FUNCTION_BLOCK FB_IndexedSiliconeMachine
VAR

    // =====================================================
    // CORE COMPONENTS
    // =====================================================
    fbIndex                     : FB_IndexTable4;
    fbMainDoorLock              : FB_MainDoorLock;
    fbNestManager               : FB_NestTableManager;
    fbOperatorStation           : FB_OperatorStation;
    

    // =====================================================
    // PROCESS COMPONENTS
    // =====================================================
    fbProcessStation            : FB_ProcessStation;
    fbProcessCycle              : FB_ProcessCycle;

    fbSiliconeProcess           : FB_SiliconeProcess;
    fbAssemblyStation           : FB_AssemblyStation;

    fbIvek                      : FB_IvekDigiSpense4000;
    fbIvekSettingsLauncher      : FB_IvekSettingsLauncher;

    ipEquipment                 : I_ProcessEquipment;

	// =====================================================
    // SILICONE SUPPLY 
    // =====================================================
	fbSiliconeSupply       : FB_SiliconeSupplySystem;
	stSiliconeSupplyStatus : ST_SiliconeSupplyStatus;
	stSiliconeSupplyConfig : ST_SiliconeSupplyConfig;
	
    // =====================================================
    // SUPPORT COMPONENTS
    // =====================================================
    fbSiliconeSupportCylinder   : FB_Support;
    fbAssemblySupportCylinder   : FB_Support;

    // =====================================================
    // MACHINE MODES
    // =====================================================
    fbManualMode                : FB_ManualMode;
	bManualAssemblySupportRaised : BOOL;

    // =====================================================
    // MACHINE / CYCLE STATES
    // =====================================================
    eMachineState               : E_MachineState := E_MachineState.PowerUp;
    ePreviousMachineState       : E_MachineState := E_MachineState.PowerUp;
    eCycleState                 : E_CycleState := E_CycleState.Disabled;

    bMachineStateEntry          : BOOL;

    eInitialisingWaitReason     : E_InitialisingWaitReason :=
                                    E_InitialisingWaitReason.None;

    eStoppingWaitReason         : E_StoppingWaitReason :=
                                    E_StoppingWaitReason.None;

    // =====================================================
    // NEST DATA
    // =====================================================
    stOperatorNest              : ST_Nest;
    stSiliconeNest              : ST_Nest;
    stAssemblyNest              : ST_Nest;
    stProcessNest               : ST_Nest;
	stFaultNest 				: ST_Nest;

    stLastResult                : ST_ProcessResult;
	bDisabledNestPartPresent 	: BOOL;

    // =====================================================
    // COMPONENT STATUS
    // =====================================================
    stOperatorStatus            : ST_OperatorStationStatus;
    stIndexStatus               : ST_IndexStatus;
    stProcessStationStatus      : ST_ProcessStationStatus;
    stAssemblyStationStatus     : ST_AssemblyStationStatus;
    stMainDoorLockStatus        : ST_MainDoorLockStatus;
	uiResetStatisticsNestIdOld 	: UINT;
	

    // =====================================================
    // MACHINE PERMISSIVES / OUTPUTS
    // =====================================================
    stPermissives               : ST_MachinePermissives;
    stOutputsInternal           : ST_MachineOutputs;
	stFaultRejectResult 		: ST_ProcessResult;
    // =====================================================
    // PROCESS CYCLE INTERFACE
    // =====================================================
    stProcessCycleInputs        : ST_ProcessCycleInputs;
    stProcessCycleRequests      : ST_ProcessCycleRequests;
    stProcessCycleStatus        : ST_ProcessCycleStatus;

    // =====================================================
    // MANUAL MODE INTERFACE
    // =====================================================
    stManualModeInputs          : ST_ManualModeInputs;
    stManualModeRequests        : ST_ManualModeRequests;
    stManualModeStatus          : ST_ManualModeStatus;

    // =====================================================
    // SUPPORT COMMANDS
    // =====================================================
    bSiliconeSupportRaiseRequest  : BOOL;
    bSiliconeSupportLowerRequest  : BOOL;

    bAssemblySupportRaiseRequest  : BOOL;
    bAssemblySupportLowerRequest  : BOOL;

    // =====================================================
    // INDEX COMMAND / FEEDBACK
    // =====================================================
    bManualIndexRequestAccepted             : BOOL;
    bManualAssemblyCycleActive                : BOOL;
    bManualSiliconeCycleActive                 : BOOL;
    bIndexRequestAcceptedFeedback           : BOOL;
    bIndexRecoveryRequestAcceptedFeedback   : BOOL;

    bIndexStable                            : BOOL;
    bIndexDone                              : BOOL;

    // =====================================================
    // PROCESS COMMAND / FEEDBACK
    // =====================================================
    bProcessStartPulse            : BOOL;
    bProcessReady                 : BOOL;
    bResultStoredFeedback         : BOOL;
    bIvekOperationPermissive      : BOOL;
    bIvekMaintenancePermissive    : BOOL;
    bIvekOperationalHealthy       : BOOL;
    bIvekAutoCycleReady           : BOOL;
    bIvekUnexpectedNotReady       : BOOL;
    tonIvekInitialisingRecovery   : TON;
    tonIvekReferenceStable        : TON;
    tonIvekUnexpectedNotReady     : TON;
    tonIvekCommunicationStop      : TON;
    tonIvekReferenceStop          : TON;

    bProcExtend                   : BOOL;
    bProcRetract                  : BOOL;

	bSiliconeProcessPartVacuumEnable : BOOL;
	bPartVacuumReleasePending        : BOOL;
	bSiliconeProcessAirEnable 		 : BOOL;
    // =====================================================
    // INITIALISATION / STOPPING
    // =====================================================
    bInitialisationComplete       : BOOL;
    bStoppingComplete             : BOOL;

    bInitialisationTimeoutFault   : BOOL;
    bStoppingTimeoutFault         : BOOL;
	bStopRequestTimeout 		  : BOOL;
	
	bExtractorAutoCycleFault 	  : BOOL;
	
    tonInitialising               : TON;
	tonInitialisingMinTime 	      : TON;
    tonStopping                   : TON;
    tonAutoCycleIdleTimeout       : TON;
	tonMainDoorNotClosed 		  : TON;
	tonStopRequest 				  : TON;
	
	
	bStopRequested 				  : BOOL;
    // =====================================================
    // AIR / DOOR CONTROL
    // =====================================================
    bAirAndDoorEnable             : BOOL;
    bAirSupplyLatched             : BOOL;
    bAirSupplyEnable              : BOOL;

    // =====================================================
    // SAFETY / FAULT HANDLING
    // =====================================================
    bSafetyDropRequest            : BOOL;

    fbEventFaultTrigger           : R_TRIG;
    fbResetTrigger                : R_TRIG;
	bFaultResetRequested 		  : BOOL;

    tpSafetyRunDrop               : TP;
	bHmiLogoutFault 				: BOOL;
		
	bSiliconePressureFault 			: BOOL;
	bNozzlePressureFault   			: BOOL;

	bSiliconePressureConfigRequired : BOOL;
	bNozzlePressureConfigRequired   : BOOL;
    // =====================================================
    // CONFIGURATION
    // =====================================================
    bConfigured                   : BOOL;
	
	// =====================================================
    // LEDS
    // =====================================================
	eMode_LED_Start 				: E_LEDs_Mode := E_LEDs_Mode.OFF;
	eMode_LED_Reset 				: E_LEDs_Mode := E_LEDs_Mode.OFF;
	eMode_LED_PASS  				: E_LEDs_Mode := E_LEDs_Mode.OFF;
	eMode_LED_Fail  				: E_LEDs_Mode := E_LEDs_Mode.OFF;

	tonLedBlink    					: TON;
	bLedBlink      					: BOOL;
	fbLedBlinkTrigger 				: R_TRIG;
	bLedBlinkState 					: BOOL;
	
	uiHistoryNestId 				: UINT;
	bHistoryPassed  				: BOOL;
	stHistoryNest   				: ST_Nest;
	// =====================================================
    // Extractor
    // =====================================================
	bExtractorEnable 				: BOOL;
	
	// CSV cycle data
	stCycleDataCSV      			: ST_CycleDataCSV;
	bCycleDataCSVWrite  			: BOOL;

END_VAR

METHOD CheckComponentFaults : BOOL
// =========================================================
// COMPONENT FAULT AGGREGATION
// =========================================================

CheckComponentFaults := FALSE;

IF fbMainDoorLock.IsFaulted()
    OR fbIndex.IsFaulted()
	OR fbSiliconeSupportCylinder.IsFaulted()
	OR fbAssemblySupportCylinder.IsFaulted()
    OR fbAssemblyStation.IsFaulted()
    OR fbProcessStation.IsFaulted()

    // Enable after equipment commissioning.
    // OR ipEquipment.IsFaulted()
THEN

    bSafetyDropRequest := TRUE;
    eMachineState := E_MachineState.Fault;

    CheckComponentFaults := TRUE;

END_IF
END_METHOD

METHOD PUBLIC Cyclic
VAR_INPUT
    stInputs       : ST_MachineInputs;
    stCommand      : ST_MachineCommand;
    stConfig       : ST_MachineConfig;
    stIvekInput    : ST_IvekCyclicInput;
    bIvekCommsOk   : BOOL;
	blogoutHMI	   : BOOL;

	
END_VAR
VAR_OUTPUT
    stOutputs      : ST_MachineOutputs;
    stStatus       : ST_MachineStatus;
    stIvekOutput   : ST_IvekCyclicOutput;
	stCycleDataCSVOut     : ST_CycleDataCSV;
	bCycleDataCSVWriteOut : BOOL;
END_VAR
// =========================================================
// GLOBAL MACHINE FAULT CONDITION
// =========================================================
// Any loss of the validated TwinSAFE safety status must place
// the machine in Fault immediately, regardless of machine state.
// =========================================================

IF NOT stInputs.stSafety.bSafetyOk OR bSafetyDropRequest THEN

    eMachineState := E_MachineState.Fault;

END_IF

// =========================================================
// MACHINE STOP REQUEST LATCH
// =========================================================

// Memorise the Stop command until the machine has
// completed the required stopping sequence.
IF (stCommand.bStop OR stCommand.bPowerDownRequest)
    AND (eMachineState <> E_MachineState.Stopping)
    AND (eMachineState <> E_MachineState.Stopped)
THEN
    bStopRequested := TRUE;
END_IF

// =========================================================
// LED BLINK GENERATOR
// =========================================================

tonLedBlink(
    IN := NOT tonLedBlink.Q,
    PT := T#500MS
);

fbLedBlinkTrigger(
    CLK := tonLedBlink.Q
);

IF fbLedBlinkTrigger.Q THEN
    bLedBlinkState := NOT bLedBlinkState;
END_IF

bLedBlink := bLedBlinkState;
// =========================================================
// DETERMINISTIC CYCLIC INITIALISATION
// =========================================================

// Deterministic defaults
ResetCyclicOutputs();

// CSV write request is generated for one PLC scan
bCycleDataCSVWrite := FALSE;

// This request is generated for one PLC scan by an internal machine fault.
// The TP converts the one-scan request into the required TwinSAFE run-drop time.
bSafetyDropRequest := FALSE;
bMachineStateEntry := eMachineState <> ePreviousMachineState;
ePreviousMachineState := eMachineState;
fbResetTrigger(
    CLK := stCommand.bReset
);

IF fbResetTrigger.Q THEN
    fbSiliconeProcess.RequestReset();
    fbAssemblyStation.RequestReset();
END_IF

fbSiliconeSupply.Cyclic(
    bLevel1Ok := stInputs.bSiliconeMinimumLevel1,
    bLevel2Ok := stInputs.bSiliconeMinimumLevel2,
    rSiliconePressureBar := stInputs.rSiliconePressureBar,
    rNozzlePressureBar := stInputs.rNozzlePressureBar,
    rVacuumEngineering := stInputs.rVacuumEngineering,

    stConfig := GVL_Config.stMachine.stSiliconeSupply,

    bCmdSelectReservoir1 := GVL_SiliconeSupply_Interface.bCmdSelectReservoir1,
    bCmdSelectReservoir2 := GVL_SiliconeSupply_Interface.bCmdSelectReservoir2,
    bCmdStartDegassing1 := GVL_SiliconeSupply_Interface.bCmdStartDegassing1,
    bCmdStartDegassing2 := GVL_SiliconeSupply_Interface.bCmdStartDegassing2,
    bCmdCancelDegassing := GVL_SiliconeSupply_Interface.bCmdCancelDegassing,
    bManualSelectionAllowed := eMachineState = E_MachineState.Stopped,

    bDispenseActive := fbSiliconeProcess.IsBusy() OR fbIvek.IsFluidicActive(),
    bDispenseValveRequest := fbSiliconeProcess.GetPinchValveRequest() OR fbIvek.IsFluidicActive(),
    bImmediateFault := eMachineState = E_MachineState.Fault,

    stPersistent := GVL_Persistent.stSiliconeSupply,

    bVacuumPump => stOutputsInternal.bVacuumPumpEnable,
    bVacuumToAir1 => stOutputsInternal.bVacuumAirSolenoid1,
    bVacuumToAir2 => stOutputsInternal.bVacuumAirSolenoid2,
    bPinchValve1 => stOutputsInternal.bSiliconePinchValve1,
    bPinchValve2 => stOutputsInternal.bSiliconePinchValve2
);

stSiliconeSupplyStatus := fbSiliconeSupply.GetStatus();
GVL_SiliconeSupply_Interface.stStatus := stSiliconeSupplyStatus;
stStatus.stSiliconeSupply := stSiliconeSupplyStatus;

IF fbSiliconeSupply.HasStopRequest() THEN
    bStopRequested := TRUE;
END_IF

IF eMachineState = E_MachineState.AutoCycle
AND stSiliconeSupplyStatus.bReservoirSelectionRequired THEN
    bStopRequested := TRUE;
END_IF

// Loss of IVEK reference is a recoverable stop condition, not an Immediate
// Fault. Stop the active machine and require Engineer Reference in Settings.
IF fbIvek.IsReferenceRequired()
AND (eMachineState = E_MachineState.AutoCycle OR eMachineState = E_MachineState.Manual) THEN
    bStopRequested := TRUE;
END_IF

// The Assembly Station is executed with its physical I/O in the component section below.

bProcessStartPulse := FALSE;

// Automatic door-lock request. Air supply is managed independently by the machine states below.
bAirAndDoorEnable := (eMachineState = E_MachineState.Initialising) OR (eMachineState = E_MachineState.ReadyToStart) OR (eMachineState = E_MachineState.AutoCycle) OR (eMachineState = E_MachineState.Manual);

stIndexStatus := fbIndex.GetStatus();
bIndexStable := NOT stIndexStatus.bBusy AND stInputs.bIndexReady AND stInputs.bIndexLocked AND stInputs.eIndexPosition <> E_TablePosition.Unknown;
bIndexDone := fbIndex.IsDone();

// =========================================================
// HMI LOGOUT SUPERVISION
// =========================================================
//
// If the HMI heartbeat is lost while the machine is already
// Stopped, the machine must remain Stopped.
//
// If the heartbeat is lost in any other operating state,
// the machine enters Fault immediately.
//
// Fault is never overridden by the HMI logout condition.
// =========================================================


// Loss of HMI heartbeat also requests a controlled stop.
// Fault has higher priority and is handled separately.
IF blogoutHMI
    AND (eMachineState = E_MachineState.Stopped OR eMachineState = E_MachineState.Stopping)THEN
	bStopRequested := TRUE;
	
ELSIF blogoutHMI
    AND (eMachineState <> E_MachineState.Stopped AND eMachineState <> E_MachineState.Stopping)THEN 
	bHmiLogoutFault := TRUE;
    bSafetyDropRequest := TRUE;
END_IF




// =========================================================
// PROCESS EQUIPMENT CONFIGURATION / CYCLIC EXECUTION
// =========================================================

// Configure the real IVEK process equipment once.
IF NOT bConfigured THEN

    ipEquipment := fbIvek;

    fbProcessStation.Configure(
        ipNewEquipment := ipEquipment
    );

    bConfigured := TRUE;

END_IF


// ---------------------------------------------------------
// IVEK machine-level operation permissive
// ---------------------------------------------------------
// Runtime motion is allowed only while:
// - EtherNet/IP communication is healthy;
// - process safety is permitted;
// - machine air is validated;
// - the machine is in AutoCycle or Manual;
// - the machine is not in Fault.
//
// FB_IvekDigiSpense4000 performs the controlled Stop-before-
// MotionDisable behaviour if this permissive is removed while
// Production is active.
bIvekOperationPermissive :=
    bIvekCommsOk
    AND stInputs.stSafety.bProcessSafetyPermitted
    AND GVL_Safety.bAirSupplySafe
    AND eMachineState <> E_MachineState.Fault
    AND (
        eMachineState = E_MachineState.Initialising
        OR eMachineState = E_MachineState.ReadyToStart
        OR eMachineState = E_MachineState.AutoCycle
        OR eMachineState = E_MachineState.Manual
    );

// Engineer Settings operations are only permitted while Stopped with the
// process safety circuit and pneumatic supply healthy.
bIvekMaintenancePermissive :=
    bIvekCommsOk
    AND (eMachineState = E_MachineState.Stopped)
    AND stInputs.stSafety.bProcessSafetyPermitted
    AND GVL_Safety.bAirSupplySafe
    AND stInputs.bMainDoorClosed;
	
stStatus.bIvekClearFaultPermissive :=
    bIvekCommsOk
    AND (eMachineState = E_MachineState.Stopped OR eMachineState = E_MachineState.Fault)
    AND fbIvek.IsFaulted();


// Always execute the real IVEK object for communication diagnostics,
// even while process simulation is selected.
fbIvek.stCyclicIn := stIvekInput;
fbIvek.bCommunicationOk := bIvekCommsOk;
fbIvek.bOperationPermissive := bIvekOperationPermissive;
fbIvek.bSystemInitialising := (eMachineState = E_MachineState.Initialising);
fbIvek.bMaintenancePermissive := bIvekMaintenancePermissive;
fbIvek.bPrimePermissive :=
    (eMachineState = E_MachineState.Manual)
    AND bIvekCommsOk
    AND stInputs.stSafety.bProcessSafetyPermitted
    AND GVL_Safety.bAirSupplySafe;
fbIvek.Cyclic();

// =========================================================
// IVEK OPERATIONAL INTERLOCK
// =========================================================
// ReadyProduction is expected to drop during a valid dispense, therefore
// permanent health is evaluated separately from start readiness.
bIvekOperationalHealthy :=
    bIvekCommsOk
    AND NOT fbIvek.IsFaulted()
    AND NOT fbIvek.IsReferenceRequired();

bIvekAutoCycleReady :=
    bIvekOperationalHealthy
    AND fbIvek.bReadyProduction
    AND NOT fbIvek.IsFluidicActive()
    AND NOT fbIvek.IsReferenceActive();

// ReadyProduction=FALSE is abnormal only while the process is idle.
// This avoids treating a normal dispense as "not ready".
bIvekUnexpectedNotReady :=
    bIvekOperationalHealthy
    AND (eMachineState <> E_MachineState.Initialising)
    AND NOT fbIvek.bReadyProduction
    AND NOT fbIvek.IsBusy()
    AND NOT fbSiliconeProcess.IsBusy()
    AND NOT fbIvek.IsFluidicActive()
    AND NOT fbIvek.IsReferenceActive();

// ReadyProduction can briefly drop around a legitimate Production transition.
// Do not stop the whole machine on a one-scan / short transient.
// Communication loss, IVEK Fault and Reference Required remain immediate
// operational-stop conditions through bIvekOperationalHealthy.
// Transient IVEK conditions must not stop the machine immediately.
// Actual IVEK faults remain immediate; communication, reference-required
// and generic not-ready are debounced to tolerate short status gaps.
tonIvekUnexpectedNotReady(
    IN := bIvekUnexpectedNotReady,
    PT := T#3S
);

tonIvekCommunicationStop(
    IN := NOT bIvekCommsOk
        AND (
            eMachineState = E_MachineState.ReadyToStart
            OR eMachineState = E_MachineState.AutoCycle
            OR eMachineState = E_MachineState.Manual
        ),
    PT := T#2S
);

tonIvekReferenceStop(
    IN := bIvekCommsOk
        AND fbIvek.IsReferenceRequired()
        AND (
            eMachineState = E_MachineState.ReadyToStart
            OR eMachineState = E_MachineState.AutoCycle
            OR eMachineState = E_MachineState.Manual
        ),
    PT := T#2S
);

// Engineer Settings commands. HMI page access is Engineer-only; PLC also
// enforces Stopped + safety/air conditions before the FB accepts motion.
// Controlled IVEK stop before PLC shutdown or reboot.
IF stCommand.bIvekMaintenanceStop THEN
    fbIvek.RequestStop();
END_IF

IF stCommand.bPowerDownRequest THEN

    // Stop active equipment/process sequences before PLC shutdown or reboot.
    fbIvek.RequestStop();
    fbSiliconeProcess.RequestStop();
    fbAssemblyStation.RequestStop();
	bStopRequested := TRUE;

END_IF

IF stCommand.bIvekReference THEN
    fbIvek.RequestReference();
END_IF

IF stCommand.bIvekClearFault THEN
    fbIvek.RequestReset();
END_IF



// Process simulation removed from runtime path. The real IVEK is always used.


IF stCommand.usiRecipeRequest <> 0 THEN
    ipEquipment.SetRecipe(stCommand.usiRecipeRequest);
END_IF


// =========================================================
// SILICONE PROCESS COORDINATOR
// =========================================================
// Execute exactly once per PLC scan, after the selected process
// equipment has updated its status for this scan.
fbSiliconeProcess.Cyclic(
    bSupplyReady 				:= fbSiliconeSupply.IsReadyForDispense(),
    bEquipmentReady 			:= fbIvek.IsReady(),
    bEquipmentBusy 				:= fbIvek.IsBusy(),
    bEquipmentDone 				:= fbIvek.IsDone(),
    bEquipmentFaulted 			:= fbIvek.IsFaulted(),
    stEquipmentResult 			:= fbIvek.GetResult(),
    bSiliconeSupportExtended 	:= stInputs.bSiliconeSupportExtended,
    bExtractorReady 			:= stPermissives.bExtractorReady,
	bPartVacuumOk 				:= stInputs.bPartVacuumOk,
	tPartVacuumBuildTimeout 	:= GVL_Config.stMachine.tPartVacuumBuildTimeout,
	tPartVacuumReleaseTimeout 	:= GVL_Config.stMachine.tPartVacuumReleaseTimeout,
    tPinchSettlingDelay 		:= GVL_Config.stMachine.stSiliconeSupply.tPinchValveSettlingDelay,
    tEquipmentStartTimeout 		:= GVL_Config.stMachine.stSiliconeSupply.tIvekStartTimeout,
    tEquipmentCompleteTimeout 	:= GVL_Config.stMachine.stSiliconeSupply.tIvekCompleteTimeout,
	bSiliconeStationPartPresent := stInputs.bSiliconeStationPartPresent,
    bPartVacuumEnable 			=> bSiliconeProcessPartVacuumEnable,
	bSiliconeAirEnable 			=> bSiliconeProcessAirEnable
);

// The coordinator generates one-scan equipment requests.
// The equipment object latches these requests and executes them
// on its next Cyclic() call.
IF fbSiliconeProcess.GetEquipmentStopRequest() THEN
    fbIvek.RequestStop();
END_IF

IF fbSiliconeProcess.GetEquipmentResetRequest() THEN
    fbIvek.RequestReset();
END_IF

IF fbSiliconeProcess.GetEquipmentStartRequest() THEN
    fbIvek.RequestStart();
END_IF

stStatus.rIvekHeaterTemperature :=
    stInputs.rIvekHeaterTemperature;

stStatus.bIvekHeaterTemperatureOutOfRange :=
    (stInputs.rIvekHeaterTemperature <
        GVL_Config.stMachine.stSiliconeSupply.rIvekHeaterTemperatureMin)
    OR
    (stInputs.rIvekHeaterTemperature >
        GVL_Config.stMachine.stSiliconeSupply.rIvekHeaterTemperatureMax);

stStatus.eIvekStatusState := fbIvek.GetStatusState();

// =========================================================
// NEST MANAGEMENT

fbNestManager.Cyclic(
    bIndexStable := bIndexStable,
    bIndexComplete := bIndexDone,

    eIndexPosition := stInputs.eIndexPosition,

    bGearboxAssemblyPartPresent := stInputs.bGearboxAssemblyPartPresent,
    bReservoirPartPresent := stInputs.bReservoirPartPresent,
    eOperatorPosition := stConfig.eOperatorPosition,
    bIndexSamePositionDetected := stIndexStatus.bSamePositionDetected,
    aNestEnabled := stConfig.aNestEnabled
);


stOperatorNest := fbNestManager.GetNestAtPosition(stConfig.eOperatorPosition);
stSiliconeNest := fbNestManager.GetNestAtPosition(stConfig.eSiliconePosition);
stAssemblyNest := fbNestManager.GetNestAtPosition(stConfig.eAssemblyPosition);

// =========================================================
// DISABLED OPERATOR NEST PART DETECTION
// =========================================================
// Disabled nests keep the existing machine behaviour while empty.
// If a part is physically detected at the operator station while
// the current operator nest is disabled, indexing will be inhibited.

bDisabledNestPartPresent :=
    NOT stOperatorNest.bEnabled
    AND
    (
        stInputs.bGearboxAssemblyPartPresent
        OR stInputs.bReservoirPartPresent
    );

// =========================================================
// MANUAL MODE - NEW PART / NEST RESULT RESET
// =========================================================
// A newly loaded part in Manual mode starts a new process history for
// the physical nest. Clear Silicone / Assembly / final results left by
// the previous part.
//
// AutoCycle keeps its existing PASS/FAIL disposition-based clear logic.
IF (eMachineState = E_MachineState.Manual)
AND stOperatorNest.bPartLoadedPulse THEN

    fbNestManager.ClearOperatorNest(
        ePosition := stConfig.eOperatorPosition
    );

    // Refresh the local snapshot after clearing the internal nest data.
    stOperatorNest :=
        fbNestManager.GetNestAtPosition(stConfig.eOperatorPosition);

END_IF

// =========================================================
// RESET CURRENT NEST STATISTICS
// =========================================================

IF stCommand.uiResetStatisticsNestId >= 1
    AND stCommand.uiResetStatisticsNestId <= 4
    AND stCommand.uiResetStatisticsNestId <> uiResetStatisticsNestIdOld
THEN

    fbNestManager.ResetNestStatistics(
        uiNestId := stCommand.uiResetStatisticsNestId
    );

END_IF

uiResetStatisticsNestIdOld :=stCommand.uiResetStatisticsNestId;

fbNestManager.CountStatisticsAtPosition(
    ePosition := stConfig.eOperatorPosition
);



// =========================================================
// TEST HISTORY EVENT
// =========================================================

IF fbNestManager.GetStatisticsEvent(
    uiNestId => uiHistoryNestId,
    bPassed  => bHistoryPassed
) THEN

    // Get the complete nest data at the moment
    // the result is added to the statistics.
    stHistoryNest := fbNestManager.GetNestAtPosition( stConfig.eOperatorPosition );


    // -----------------------------------------------------
    // STORE TEST HISTORY ENTRY
    // -----------------------------------------------------

    GVL_Persistent.astTestHistory[GVL_Persistent.uiTestHistoryWriteIndex].uiNestId 				:= uiHistoryNestId;
    GVL_Persistent.astTestHistory[GVL_Persistent.uiTestHistoryWriteIndex].eResult 				:= stHistoryNest.eDisposition;
    GVL_Persistent.astTestHistory[GVL_Persistent.uiTestHistoryWriteIndex].bSiliconeValid 		:= stHistoryNest.stSiliconeResult.bValid;
    GVL_Persistent.astTestHistory[GVL_Persistent.uiTestHistoryWriteIndex].bSiliconePass 		:= stHistoryNest.stSiliconeResult.bPassed;
    GVL_Persistent.astTestHistory[GVL_Persistent.uiTestHistoryWriteIndex].bAssemblyValid 		:= stHistoryNest.stAssemblyResult.bValid;
    GVL_Persistent.astTestHistory[GVL_Persistent.uiTestHistoryWriteIndex].bAssemblyPass 		:= stHistoryNest.stAssemblyResult.bPassed;
	GVL_Persistent.astTestHistory[GVL_Persistent.uiTestHistoryWriteIndex].sDate 				:= GVL_MASTER.sSystemDate;
	GVL_Persistent.astTestHistory[GVL_Persistent.uiTestHistoryWriteIndex].sTime 				:= GVL_MASTER.sSystemTime;
				
				// Final result text
		IF stHistoryNest.stResult.bPassed THEN
			GVL_Persistent.astTestHistory[GVL_Persistent.uiTestHistoryWriteIndex].sResult := 'PASS';
		ELSE
			GVL_Persistent.astTestHistory[GVL_Persistent.uiTestHistoryWriteIndex].sResult := 'FAIL';
		END_IF;
		
		
		// Silicone result text
		IF NOT stHistoryNest.stSiliconeResult.bValid THEN
		
			GVL_Persistent.astTestHistory[GVL_Persistent.uiTestHistoryWriteIndex].sSiliconeResult := 'NOT STARTED';
		
		ELSIF stHistoryNest.stSiliconeResult.bPassed THEN
		
			GVL_Persistent.astTestHistory[GVL_Persistent.uiTestHistoryWriteIndex].sSiliconeResult := 'PASS';
		
		ELSE
		
			GVL_Persistent.astTestHistory[GVL_Persistent.uiTestHistoryWriteIndex].sSiliconeResult := 'FAIL';
		
		END_IF;
		
		
		// Flipping result text
		IF NOT stHistoryNest.stAssemblyResult.bValid THEN
		
			GVL_Persistent.astTestHistory[GVL_Persistent.uiTestHistoryWriteIndex].sFlippingResult := 'NOT STARTED';
		
		ELSIF stHistoryNest.stAssemblyResult.bPassed THEN
		
			GVL_Persistent.astTestHistory[GVL_Persistent.uiTestHistoryWriteIndex].sFlippingResult := 'PASS';
		
		ELSE
		
			GVL_Persistent.astTestHistory[GVL_Persistent.uiTestHistoryWriteIndex].sFlippingResult := 'FAIL';
		
		END_IF;
				
		// -----------------------------------------------------
		// PREPARE CSV CYCLE DATA
		// -----------------------------------------------------
		
		stCycleDataCSV.uiNestId :=
			GVL_Persistent.astTestHistory[GVL_Persistent.uiTestHistoryWriteIndex].uiNestId;
		
		stCycleDataCSV.sGeneralResult :=
			GVL_Persistent.astTestHistory[GVL_Persistent.uiTestHistoryWriteIndex].sResult;
		
		stCycleDataCSV.sSiliconeResult :=
			GVL_Persistent.astTestHistory[GVL_Persistent.uiTestHistoryWriteIndex].sSiliconeResult;
		
		stCycleDataCSV.sFlippingResult :=
			GVL_Persistent.astTestHistory[GVL_Persistent.uiTestHistoryWriteIndex].sFlippingResult;
		
		stCycleDataCSV.sDate :=
			GVL_Persistent.astTestHistory[GVL_Persistent.uiTestHistoryWriteIndex].sDate;
		
		stCycleDataCSV.sTime :=
			GVL_Persistent.astTestHistory[GVL_Persistent.uiTestHistoryWriteIndex].sTime;
		
		bCycleDataCSVWrite := TRUE;	
				
				
				
		// -----------------------------------------------------
		// ADVANCE TEST HISTORY WRITE INDEX
		// -----------------------------------------------------
		
		IF GVL_Persistent.uiTestHistoryCount < 2001 THEN
			GVL_Persistent.uiTestHistoryCount := GVL_Persistent.uiTestHistoryCount + 1;
		END_IF
		
		IF GVL_Persistent.uiTestHistoryWriteIndex < 2000 THEN
		
			GVL_Persistent.uiTestHistoryWriteIndex := GVL_Persistent.uiTestHistoryWriteIndex + 1;
		
		ELSE
		
			GVL_Persistent.uiTestHistoryWriteIndex := 0;
		
		END_IF
		

END_IF



// =========================================================
// OPERATOR STATION CONTROL
// =========================================================


// Operator exchange is evaluated independently of process-equipment implementation.
fbOperatorStation.Cyclic(
    bAutomaticActive := eMachineState = E_MachineState.AutoCycle,
    bIndexStable := bIndexStable,
    stOperatorNest := stOperatorNest,
    bGearboxAssemblyPartPresent := stInputs.bGearboxAssemblyPartPresent,
    bReservoirPartPresent := stInputs.bReservoirPartPresent,
    bRejectChutePartPresent := stInputs.bRejectChutePartPresent,
    bRequireRejectConfirm := stConfig.bRequireRejectConfirm,
    bAllowEmptyNestIndex := stConfig.bAllowEmptyNestIndex);
	
stOperatorStatus := fbOperatorStation.GetStatus();

// =========================================================
// OPERATOR NEST RESULT RELEASE
// =========================================================


// PASS: clear after part removal.
IF stOperatorNest.stResult.bValid
    AND stOperatorNest.stResult.bPassed
    AND stOperatorStatus.bPartRemovedConfirmed
THEN

    fbNestManager.ClearOperatorNest(
        stConfig.eOperatorPosition
    );

END_IF


// FAIL: clear only after reject confirmation.
IF stOperatorNest.stResult.bValid
    AND NOT stOperatorNest.stResult.bPassed
    AND stOperatorStatus.bRejectConfirmed
THEN

    fbNestManager.ClearOperatorNest(
        stConfig.eOperatorPosition
    );

END_IF

// =========================================================
// MACHINE PERMISSIVE AGGREGATION
// =========================================================

// Explicit permissive aggregation.
stPermissives.bSafetyIndexPermissive 	:= 	stInputs.stSafety.bMotionSafetyPermitted;
stPermissives.bOperatorIndexPermissive 	:= 	fbOperatorStation.IndexPermissive();
stPermissives.bProcessIndexPermissive 	:= 	NOT fbSiliconeProcess.IsBusy()
											AND NOT fbSiliconeProcess.IsFaulted()
											AND fbAssemblyStation.IndexPermissive();

stPermissives.bIndexMoveAllowed :=
											stPermissives.bSafetyIndexPermissive
											//AND stPermissives.bOperatorIndexPermissive
											AND stPermissives.bProcessIndexPermissive
											AND NOT bDisabledNestPartPresent;


stPermissives.bProcessStartAllowed 		:= 	stInputs.stSafety.bProcessSafetyPermitted
											AND stInputs.bIndexReady
											AND stInputs.bIndexLocked
											AND stInputs.bReservoirPartPresent;
											
stPermissives.bExtractorReady 			:=  stInputs.bExtractorRunning;


// =========================================================
// INITIALISATION PERMISSIVES
// =========================================================

stPermissives.bAirSupplyReady :=
	GVL_Safety.bAirSupplySafe;

stPermissives.bSiliconeSupportHome :=
    stInputs.bSiliconeSupportRetracted;

stPermissives.bAssemblySupportHome :=
    stInputs.bAssemblySupportRetracted;

stPermissives.bSupportsHome :=
    stPermissives.bSiliconeSupportHome
    AND stPermissives.bAssemblySupportHome;

stPermissives.bAssemblyStationHome := fbAssemblyStation.IsHome();

stPermissives.bIndexInitialisationReady :=
    ( NOT stIndexStatus.bBusy
        OR
        (stIndexStatus.eState = E_IndexState.WrongPositionRecovery
            AND stInputs.eIndexPosition = E_TablePosition.Unknown)
    )
    AND NOT fbIndex.IsFaulted();

stPermissives.bDoorInitialisationReady :=
    NOT fbMainDoorLock.IsFaulted()
    AND fbMainDoorLock.IsReadyForAutomatic();

stPermissives.bInitialisationAllowed :=
    stInputs.stSafety.bSafetyOk
    AND stPermissives.bAirSupplyReady
    AND stPermissives.bIndexInitialisationReady
    AND stPermissives.bSupportsHome
    AND stPermissives.bAssemblyStationHome
    AND NOT fbAssemblyStation.IsFaulted()
    AND stPermissives.bDoorInitialisationReady
    AND stPermissives.bExtractorReady
    AND NOT stInputs.bIvekHeaterControllerAlarm
	AND NOT stStatus.bIvekHeaterTemperatureOutOfRange ;
	//AND stSiliconeSupplyStatus.bSiliconePressureOk
    //AND stSiliconeSupplyStatus.bNozzlePressureOk;
	

// =========================================================
// IVEK NATIVE SETTINGS LAUNCHER
// =========================================================
 
fbIvekSettingsLauncher(
    bOpenRequest 		:= GVL_HMI.bCmdOpenIvekSettings,
    bMachineStopped 	:= eMachineState = E_MachineState.Stopped,
    udiLauncherHeartbeat := GVL_HMI.udiIvekSettingsHeartbeat,
    bResetError 		:= stCommand.bReset,
    bLauncherActive 	:= GVL_HMI.bIvekSettingsActive,
    bOpenPermitted 		=> GVL_HMI.bIvekSettingsAccessAllowed,
    bSettingsInterlock 	=> GVL_HMI.bIvekSettingsInterlock,
    bLaunchPending 		=> GVL_HMI.bIvekSettingsLaunchPending,
    bLaunchBusy 		=> GVL_HMI.bIvekSettingsLaunchBusy,
    bLaunchError 		=> GVL_HMI.bIvekSettingsLaunchError,
    nLaunchErrorId 		=> GVL_HMI.nIvekSettingsLaunchErrorId,
    bActivationTimeout 	=> GVL_HMI.bIvekSettingsActTimeout,
    bHeartbeatLost 		=> GVL_HMI.bIvekSettingsHeartbeatLost
);

// =========================================================
// EVENT ARCHITECTURE NOTES
// =========================================================

// Event architecture from the Leak Tester.
// Point classification is fixed in PRG_Events; station latches are provided
// through stInputs.bEventFault and stInputs.bEventCycleStopRequest.

// =========================================================
// MANUAL MODE COORDINATOR
// =========================================================

// Manual-mode coordinator consumes only normalized component status and produces requests.
stManualModeInputs.bSafetyOk 						:= stInputs.stSafety.bSafetyOk;
stManualModeInputs.bMotionSafetyPermitted 			:= stInputs.stSafety.bMotionSafetyPermitted;
stManualModeInputs.bTwoHandsSafe 					:= stInputs.bTwoHandsSafe;
stManualModeInputs.bProcessSafetyPermitted 			:= stInputs.stSafety.bProcessSafetyPermitted;
stManualModeInputs.bMainDoorSafe 					:= stInputs.stSafety.bMainDoorSafe;
stManualModeInputs.bIndexReady 						:= stInputs.bIndexReady;
stManualModeInputs.bIndexLocked 					:= stInputs.bIndexLocked;
stManualModeInputs.bIndexBusy 						:= stIndexStatus.bBusy;
stManualModeInputs.bIndexFaulted 					:= fbIndex.IsFaulted();
stManualModeInputs.bSiliconeSupportExtended 		:=stInputs.bSiliconeSupportExtended;
stManualModeInputs.bSiliconeSupportRetracted 		:=stInputs.bSiliconeSupportRetracted;
stManualModeInputs.bAssemblySupportExtended 		:=stInputs.bAssemblySupportExtended;
stManualModeInputs.bAssemblySupportRetracted 		:=stInputs.bAssemblySupportRetracted;



stManualModeInputs.bProcessStationFaulted := fbProcessStation.IsFaulted();
stManualModeInputs.bEquipmentReady := fbIvek.IsReady();
stManualModeInputs.bEquipmentBusy := fbIvek.IsBusy();
stManualModeInputs.bEquipmentFaulted := fbIvek.IsFaulted();

stManualModeInputs.bIvekEnabled := bIvekCommsOk AND NOT fbIvek.bMotionDisabled;
stManualModeInputs.bIvekFluidicReady := fbIvek.IsFluidicReady();
stManualModeInputs.bIvekFluidicActive := fbIvek.IsFluidicActive();
stManualModeInputs.bPartVacuumOk := stInputs.bPartVacuumOk;
stManualModeInputs.bIvekPrimeEnable :=stCommand.bIvekPrimeEnable;
stManualModeInputs.bNozzlePressureOk :=stSiliconeSupplyStatus.bNozzlePressureOk;

stManualModeInputs.bSiliconeProcessReady := fbSiliconeProcess.IsReady();
stManualModeInputs.bSiliconeProcessBusy := fbSiliconeProcess.IsBusy();
stManualModeInputs.bSiliconeProcessFaulted := fbSiliconeProcess.IsFaulted();
stManualModeInputs.bSiliconeNestPartPresent := stSiliconeNest.bPartComplete;
stManualModeInputs.bSiliconeNestAlreadyProcessed :=
    stSiliconeNest.stSiliconeResult.bValid;

stManualModeInputs.bReservoirPartPresent :=stInputs.bSiliconeStationPartPresent;
stManualModeInputs.bAssemblyStationReady := fbAssemblyStation.IsReady();
stManualModeInputs.bAssemblyStationBusy := fbAssemblyStation.IsBusy();
stManualModeInputs.bAssemblyStationFaulted := fbAssemblyStation.IsFaulted();
stManualModeInputs.bAssemblyNestPartPresent := stAssemblyNest.bPartComplete;
stManualModeInputs.bAssemblyNestSiliconized :=
    stAssemblyNest.stSiliconeResult.bValid
    AND stAssemblyNest.stSiliconeResult.bPassed;
stManualModeInputs.bAssemblyNestAlreadyAssembled :=
    stAssemblyNest.stAssemblyResult.bValid;

fbManualMode.Cyclic(
    bEnable := eMachineState = E_MachineState.Manual,
    bStopRequest := bStopRequested,
    stCommand := stCommand,
    stInputs := stManualModeInputs,
    stRequests => stManualModeRequests,
    stStatus => stManualModeStatus);
	
	
// =========================================================
// SILICONE AIR OUTPUT ARBITRATION
// =========================================================

stOutputsInternal.bSiliconeAirEnable :=
    bSiliconeProcessAirEnable
    OR (
        (eMachineState = E_MachineState.Manual)
        AND stManualModeRequests.bSiliconeAirEnable
    );
	
	
// =========================================================
// PART VACUUM RELEASE CONFIRMATION
// =========================================================

// Latch the release condition when a process has finished
// while vacuum is still present, or when Manual Prime
// explicitly requests vacuum release.
IF (fbSiliconeProcess.IsDone() AND stInputs.bPartVacuumOk)
    OR stManualModeRequests.bPartVacuumReleaseRequest
THEN
    bPartVacuumReleasePending := TRUE;
END_IF

// Release is complete only after the Silicone Support is
// fully retracted and the station is confirmed empty.
IF bPartVacuumReleasePending
    AND stInputs.bSiliconeSupportRetracted
    AND NOT stInputs.bSiliconeStationPartPresent
THEN
    bPartVacuumReleasePending := FALSE;
END_IF

// A new intentional Manual Prime vacuum request is allowed
// only after the previous release sequence has physically
// completed.
IF (eMachineState = E_MachineState.Manual)
    AND stManualModeRequests.bPartVacuumEnable
    AND stInputs.bSiliconeSupportExtended
    AND stInputs.bSiliconeStationPartPresent
THEN
    bPartVacuumReleasePending := FALSE;
END_IF	
// Allow a new Silicone process to take ownership of the vacuum
// once a new part is confirmed in the raised Silicone Support.

IF bSiliconeProcessPartVacuumEnable
    AND stInputs.bSiliconeSupportExtended
    AND stInputs.bSiliconeStationPartPresent
THEN
    bPartVacuumReleasePending := FALSE;
END_IF
	
// =========================================================
// PART VACUUM OUTPUT ARBITRATION
// =========================================================
// In automatic operation the part vacuum follows the machine
// pneumatic lifecycle while the Silicone Support is retracted.
//
// During the Silicone process, FB_SiliconeProcess owns the vacuum.
// After dispensing it removes its vacuum request before the
// Silicone Support retracts. Once the support is fully retracted,
// the normal vacuum request is restored.
//
// Manual Mode keeps its existing independent vacuum control.

stOutputsInternal.bPartVacuumEnable :=
    NOT bPartVacuumReleasePending
    AND
    (
        bSiliconeProcessPartVacuumEnable
        OR (
            bExtractorEnable
            AND stInputs.bSiliconeSupportRetracted
        )
        OR (
            (eMachineState = E_MachineState.Manual)
            AND stManualModeRequests.bPartVacuumEnable
        )
    );
// Manual Prime equipment request.
// The complete mechanical/vacuum sequence is coordinated by FB_ManualMode.
IF (eMachineState = E_MachineState.Manual)
AND stManualModeRequests.bIvekPrime THEN
    fbIvek.RequestPrime();
END_IF

stProcessCycleInputs.bSiliconeSupportExtended := stInputs.bSiliconeSupportExtended;
stProcessCycleInputs.bSiliconeSupportRetracted := stInputs.bSiliconeSupportRetracted;
stProcessCycleInputs.bAssemblySupportExtended := stInputs.bAssemblySupportExtended;
stProcessCycleInputs.bAssemblySupportRetracted := stInputs.bAssemblySupportRetracted;

// =========================================================
// STOP REQUEST TIMEOUT SUPERVISION
// =========================================================
// Once a Stop request has been latched, the machine must
// reach the Stopping state within the allowed time.
//
// This supervises the conditions that may delay leaving
// AutoCycle or Manual mode after a Stop request.
tonStopRequest(
    IN := bStopRequested
        AND eMachineState <> E_MachineState.Stopping
        AND eMachineState <> E_MachineState.Stopped
        AND eMachineState <> E_MachineState.Fault,
    PT := T#10S
);

IF tonStopRequest.Q THEN
    bStopRequestTimeout := TRUE;
    bSafetyDropRequest := TRUE;
END_IF


IF stStatus.bIvekHeaterTemperatureOutOfRange
    AND (eMachineState = E_MachineState.Manual)
THEN
    bSafetyDropRequest := TRUE;
END_IF
// =========================================================
// PRESSURE FAULT CAUSE LATCH
// =========================================================

// Pressure faults are valid only while pressure is expected.
// Once detected, keep the cause latched while the machine
// transitions to Fault.

IF
    (
        stSiliconeSupplyStatus.bSiliconePressureLow
        OR stSiliconeSupplyStatus.bSiliconePressureHigh
    )
    AND (eMachineState = E_MachineState.AutoCycle
		OR eMachineState = E_MachineState.Manual)
THEN
    bSiliconePressureFault := TRUE;
    bSafetyDropRequest := TRUE;
END_IF


IF
    (
        stSiliconeSupplyStatus.bNozzlePressureLow
        OR stSiliconeSupplyStatus.bNozzlePressureHigh
    )
    AND (eMachineState = E_MachineState.AutoCycle
		OR eMachineState = E_MachineState.Manual)
THEN
    bNozzlePressureFault := TRUE;
	bSafetyDropRequest := TRUE;
END_IF



// =========================================================
// MACHINE STATE MANAGEMENT
// =========================================================

CASE eMachineState OF
	

	E_MachineState.PowerUp:
	
		eMode_LED_Start := E_LEDs_Mode.OFF;
		eMode_LED_Reset := E_LEDs_Mode.FLASHING;
		eMode_LED_PASS  := E_LEDs_Mode.OFF;
		eMode_LED_Fail  := E_LEDs_Mode.OFF;
		
		// Air is not enabled during PowerUp or the first transition to Stopped.
		bAirSupplyEnable := FALSE;
		bExtractorEnable := FALSE;

		// Same machine lifecycle used by the Kistler: always enter a controlled stop first.
		tonInitialising(IN := FALSE);
		tonInitialisingMinTime(IN := FALSE);
		tonStopping(IN := FALSE);
		eCycleState := E_CycleState.Disabled;
		eMachineState := E_MachineState.Stopping;

	E_MachineState.Fault:

		eMode_LED_Start := E_LEDs_Mode.OFF;
		eMode_LED_Reset := E_LEDs_Mode.FLASHING;
		eMode_LED_PASS  := E_LEDs_Mode.OFF;
		eMode_LED_Fail  := E_LEDs_Mode.ON;
		
		IF bMachineStateEntry THEN

			stFaultRejectResult.bValid := TRUE;
			stFaultRejectResult.bPassed := FALSE;
			stFaultRejectResult.eCode := E_ProcessResultCode.Aborted;
			stFaultRejectResult.sDetail := 'Rejected due to machine fault';
		
			// Position 2
			stFaultNest := fbNestManager.GetNestAtPosition(E_TablePosition.Position2);
		
			IF stFaultNest.bGearboxAssemblyPartPresent OR stFaultNest.bReservoirPartPresent THEN
				fbNestManager.StoreResultAtPosition(ePosition := E_TablePosition.Position2, stResult := stFaultRejectResult);
			END_IF
		
			// Position 3
			stFaultNest := fbNestManager.GetNestAtPosition(E_TablePosition.Position3);
		
			IF stFaultNest.bGearboxAssemblyPartPresent OR stFaultNest.bReservoirPartPresent THEN
				fbNestManager.StoreResultAtPosition(ePosition := E_TablePosition.Position3, stResult := stFaultRejectResult);
			END_IF
		
			// Position 4
			stFaultNest := fbNestManager.GetNestAtPosition(E_TablePosition.Position4);
		
			IF stFaultNest.bGearboxAssemblyPartPresent OR stFaultNest.bReservoirPartPresent THEN
				fbNestManager.StoreResultAtPosition(ePosition := E_TablePosition.Position4, stResult := stFaultRejectResult);
			END_IF
		
		END_IF
		bAirSupplyEnable := FALSE;
		bExtractorEnable := FALSE;
	
		tonInitialising(IN := FALSE);
		tonInitialisingMinTime(IN := FALSE);
		tonStopping(IN := FALSE);
		fbSiliconeProcess.RequestStop();
		fbIvek.RequestStop();
		
	
		// -----------------------------------------------------
		// LATCH RESET REQUEST
		// -----------------------------------------------------
		IF fbResetTrigger.Q AND NOT blogoutHMI THEN
	
			bFaultResetRequested := TRUE;
			bHmiLogoutFault := FALSE;
			bStopRequestTimeout := FALSE;
			bExtractorAutoCycleFault := FALSE;
			bInitialisationTimeoutFault := FALSE;
    		bStoppingTimeoutFault := FALSE;
			bSiliconePressureFault := FALSE;
			bNozzlePressureFault := FALSE;
	
			fbIndex.Reset();
			fbSiliconeSupportCylinder.Reset();
			fbAssemblySupportCylinder.Reset();
            fbAssemblyStation.Reset();
	
			fbIvek.RequestReset();
	
			bInitialisationTimeoutFault := FALSE;
			bStoppingTimeoutFault := FALSE;
	
			eCycleState := E_CycleState.Disabled;
	
		END_IF


    // -----------------------------------------------------
    // LEAVE FAULT ONLY AFTER ALL COMPONENTS ARE HEALTHY
    // -----------------------------------------------------
    IF bFaultResetRequested
        AND stInputs.stSafety.bSafetyOk
        AND NOT fbIndex.IsFaulted()
        AND NOT fbSiliconeSupportCylinder.IsFaulted()
        AND NOT fbAssemblySupportCylinder.IsFaulted()
        AND NOT fbAssemblyStation.IsFaulted()
        AND NOT fbProcessStation.IsFaulted()
    THEN

        bFaultResetRequested := FALSE;

        eMachineState := E_MachineState.Stopping;

    END_IF
	
	E_MachineState.Stopping:

		tonInitialising(IN := FALSE);
		tonStopping(
			IN := TRUE,
			PT := stConfig.tStoppingTimeout
		);
	
		fbIvek.RequestStop();
	
		stIndexStatus := fbIndex.GetStatus();
	
		stMainDoorLockStatus := fbMainDoorLock.GetStatus();
	
		eStoppingWaitReason := E_StoppingWaitReason.None;
	
	
		// ---------------------------------------------------------
		// INDEX MUST BE STOPPED
		// ---------------------------------------------------------
	
		IF stIndexStatus.bBusy THEN
		eStoppingWaitReason := E_StoppingWaitReason.IndexStillMoving;
	
	
	ELSIF (stMainDoorLockStatus.eState = E_MainDoorLockState.Locking)
		OR (stMainDoorLockStatus.eState = E_MainDoorLockState.Unlocking)
	THEN
		eStoppingWaitReason := E_StoppingWaitReason.MainDoorTransition;
	END_IF
	
	
		// ---------------------------------------------------------
		// STOPPING COMPLETION
		// ---------------------------------------------------------
	
		bStoppingComplete := eStoppingWaitReason = E_StoppingWaitReason.None;
	
		IF bStoppingComplete THEN
	
			tonStopping(IN := FALSE);
	
			eCycleState := E_CycleState.Disabled;
	
			eMachineState := E_MachineState.Stopped;
	
		ELSIF tonStopping.Q THEN
	
			bStoppingTimeoutFault := TRUE;
			bSafetyDropRequest := TRUE;
				
			eMachineState := E_MachineState.Fault;
				
		END_IF
	
	E_MachineState.Stopped:
	
		eMode_LED_Start := E_LEDs_Mode.OFF;
		eMode_LED_Reset := E_LEDs_Mode.FLASHING;
		eMode_LED_PASS  := E_LEDs_Mode.OFF;
		eMode_LED_Fail  := E_LEDs_Mode.OFF;
	
		bStopRequested := FALSE;
		
		
		tonInitialising(IN := FALSE);
		tonInitialisingMinTime(IN := FALSE);
		tonStopping(IN := FALSE);
		
		IF blogoutHMI THEN
				bStopRequested := TRUE;
		ELSE
		//fbIvek.RequestStop();

			// Air may remain enabled after returning from an active machine state,
			// provided that the main door remains closed. Opening the door removes
			// the request. Closing it again does not restore the air in Stopped.
			IF NOT stInputs.bMainDoorClosed THEN
				bAirSupplyEnable := FALSE;
				bExtractorEnable := FALSE;
			END_IF
		
			IF NOT GVL_HMI.bIvekSettingsInterlock THEN
		
				IF stCommand.bReset
                    AND stInputs.stSafety.bSafetyOk
                    AND NOT fbIvek.IsFluidicActive()
                    AND NOT fbIvek.IsReferenceActive()
                THEN
					eMachineState := E_MachineState.Initialising;
				END_IF
				
			END_IF
		 END_IF
// 	
	E_MachineState.Initialising:
		// =========================================================
		// TIMERS
		// =========================================================
	
		tonStopping(IN := FALSE);
		tonInitialising(IN := TRUE, PT := stConfig.tInitialiseTimeout);
		tonInitialisingMinTime(IN := TRUE, PT := stConfig.tInitialiseMinTime);

		eMode_LED_Start := E_LEDs_Mode.OFF;
		eMode_LED_Reset := E_LEDs_Mode.OFF;
		eMode_LED_PASS := E_LEDs_Mode.OFF;
		eMode_LED_Fail := E_LEDs_Mode.OFF;

		IF NOT stInputs.bMainDoorClosed AND NOT stInputs.bMainDoorFeedback THEN
			eMachineState := E_MachineState.Fault;
		END_IF
		
		// =========================================================
		// AIR SUPPLY
		// =========================================================
		// Initialising restores the pneumatic supply before
		// recovering and validating safe component positions.
		// =========================================================
		
		bAirSupplyEnable := TRUE;
		bExtractorEnable := TRUE;
	
		// =========================================================
		// STATE ENTRY
		// =========================================================
	
		IF bMachineStateEntry THEN
	
			// fbProcessCycle.Initialise();
			// fbManualMode.Initialise();
			// fbProcessStation.Initialise();
	
			fbMainDoorLock.Initialise();
	
			// bResultStoredFeedback := FALSE;
	
			bIndexRequestAcceptedFeedback := FALSE;
			bIndexRecoveryRequestAcceptedFeedback := FALSE;
			bSiliconePressureConfigRequired := FALSE;
			bNozzlePressureConfigRequired := FALSE;
	
			// bProcessStartPulse := FALSE;
	
		END_IF
		// =========================================================
		// CURRENT COMPONENT STATUS
		// =========================================================
	
		stIndexStatus := fbIndex.GetStatus();
		stProcessStationStatus := fbProcessStation.GetStatus();
        stAssemblyStationStatus := fbAssemblyStation.GetStatus();
		stMainDoorLockStatus := fbMainDoorLock.GetStatus();
		
		
		
		
		// =========================================================
		// INITIALISING WAIT REASON
		// =========================================================
		
		eInitialisingWaitReason := E_InitialisingWaitReason.None;
		
		
		// ---------------------------------------------------------
		// AIR SUPPLY MUST BE READY
		// ---------------------------------------------------------
		
		IF NOT stPermissives.bAirSupplyReady THEN
		
			eInitialisingWaitReason := E_InitialisingWaitReason.AirSupplyNotReady;
		// ---------------------------------------------------------
		// VACUUM EXTRACTOR MUST BE RUNNING
		// ---------------------------------------------------------
		
		ELSIF NOT stPermissives.bExtractorReady THEN
		
			eInitialisingWaitReason  :=E_InitialisingWaitReason.ExtractorNotReady;
		
		ELSIF stInputs.bIvekHeaterControllerAlarm OR stStatus.bIvekHeaterTemperatureOutOfRange THEN

    		eInitialisingWaitReason := E_InitialisingWaitReason.IvekHeaterNotReady;
		
		// ---------------------------------------------------------
		// INDEX MUST NOT BE BUSY
		// ---------------------------------------------------------
		
		ELSIF stIndexStatus.bBusy THEN
		
			eInitialisingWaitReason :=
				E_InitialisingWaitReason.IndexBusy;
		
		
		// ---------------------------------------------------------
		// SILICONE SUPPORT MUST NOT BE FAULTED
		// ---------------------------------------------------------
		
		ELSIF fbSiliconeSupportCylinder.IsFaulted() THEN
		
			eInitialisingWaitReason :=
				E_InitialisingWaitReason.SiliconeSupportFaulted;
		
		
		// ---------------------------------------------------------
		// ASSEMBLY SUPPORT MUST NOT BE FAULTED
		// ---------------------------------------------------------
		
		ELSIF fbAssemblySupportCylinder.IsFaulted() THEN
		
			eInitialisingWaitReason :=
				E_InitialisingWaitReason.AssemblySupportFaulted;
		
		
		// ---------------------------------------------------------
		// SILICONE SUPPORT MUST BE RETRACTED
		// ---------------------------------------------------------
		
		ELSIF NOT stPermissives.bSiliconeSupportHome THEN
		
			eInitialisingWaitReason :=
				E_InitialisingWaitReason.SiliconeSupportNotRetracted;
		
		
		// ---------------------------------------------------------
		// ASSEMBLY SUPPORT MUST BE RETRACTED
		// ---------------------------------------------------------
		
		ELSIF NOT stPermissives.bAssemblySupportHome THEN
		
			eInitialisingWaitReason :=
				E_InitialisingWaitReason.AssemblySupportNotRetracted;
		
		
        // ---------------------------------------------------------
        // ASSEMBLY / FLIPPING STATION MUST BE HOME
        // ---------------------------------------------------------
        ELSIF fbAssemblyStation.IsFaulted() THEN

            eInitialisingWaitReason :=
                E_InitialisingWaitReason.AssemblyStationFaulted;

        ELSIF NOT stPermissives.bAssemblyStationHome THEN

            eInitialisingWaitReason :=
                E_InitialisingWaitReason.AssemblyStationNotHome;


		// ---------------------------------------------------------
		// MAIN DOOR MUST NOT BE FAULTED
		// ---------------------------------------------------------
		
		ELSIF fbMainDoorLock.IsFaulted() THEN
		
			eInitialisingWaitReason :=
				E_InitialisingWaitReason.MainDoorFaulted;
		
		
		// ---------------------------------------------------------
		// MAIN DOOR MUST BE READY FOR AUTOMATIC OPERATION
		// ---------------------------------------------------------
		
		ELSIF NOT fbMainDoorLock.IsReadyForAutomatic() THEN
		
			eInitialisingWaitReason :=
				E_InitialisingWaitReason.MainDoorNotReady;
		
		END_IF
				
		
		
		// =========================================================
		// INITIALISATION COMPLETE
		// =========================================================
	
		bInitialisationComplete := stPermissives.bInitialisationAllowed 
									AND tonInitialisingMinTime.Q;

// =========================================================
// IVEK RECOVERY DURING INITIALISING
// =========================================================
// After an Immediate Fault the IVEK communication/status can take a short
// time to recover. Do not bounce immediately back to Stopped just because
// communication / fault / ReadyProduction are still transient.
//
// Reference Required is treated separately: it must be stable for 500 ms
// before Initialising is aborted to Stopped, because the bit can briefly
// appear while the IVEK is recovering.
//
// Communication / IVEK fault / Production Ready are allowed to recover for
// up to 5 seconds. If they recover, Initialising proceeds directly to
// ReadyToStart. If not, the machine returns to Stopped with the corresponding
// persistent IVEK diagnostic remaining active.
// =========================================================

tonIvekReferenceStable(
    IN := fbIvek.IsReferenceRequired(),
    PT := T#500MS
);

tonIvekInitialisingRecovery(
    IN := bInitialisationComplete
        AND NOT bIvekAutoCycleReady
        AND NOT tonIvekReferenceStable.Q
        // LoadRequired is actively recoverable during System Initialising.
        // Do not abort after 5 s while the Load recovery is pending/running;
        // the normal machine Initialising timeout remains the final safeguard.
        AND NOT fbIvek.bLoadRequired
        AND NOT fbIvek.bLoadStartPending
        AND NOT fbIvek.bLoadRequestActive
        AND NOT fbIvek.bBusyLoad,
    PT := T#5S
);

IF bInitialisationComplete
    AND NOT stSiliconeSupplyStatus.bSelectedReservoirReady
THEN
    // Silicone supply is not ready.
    // Return to Stopped so the reservoir can be configured in Settings.
    tonIvekInitialisingRecovery(IN := FALSE);
    tonIvekReferenceStable(IN := FALSE);
    tonInitialising(IN := FALSE);
    eCycleState := E_CycleState.Disabled;
    eMachineState := E_MachineState.Stopped;

ELSIF bInitialisationComplete
    AND bIvekAutoCycleReady
THEN
    tonIvekInitialisingRecovery(IN := FALSE);
    tonIvekReferenceStable(IN := FALSE);
    tonInitialising(IN := FALSE);
    eCycleState := E_CycleState.Disabled;
    eMachineState := E_MachineState.ReadyToStart;

ELSIF bInitialisationComplete
    AND tonIvekReferenceStable.Q
THEN
    // Reference Required needs Engineer action.
    tonIvekInitialisingRecovery(IN := FALSE);
    tonInitialising(IN := FALSE);
    eCycleState := E_CycleState.Disabled;
    eMachineState := E_MachineState.Stopped;

ELSIF bInitialisationComplete
    AND tonIvekInitialisingRecovery.Q
THEN
    // Communication / IVEK fault / Not Ready did not recover in time.
    tonInitialising(IN := FALSE);
    eCycleState := E_CycleState.Disabled;
    eMachineState := E_MachineState.Stopped;

ELSIF tonInitialising.Q THEN
    bInitialisationTimeoutFault := TRUE;
    bSafetyDropRequest := TRUE;
END_IF

E_MachineState.ReadyToStart:
		

        // ReadyToStart is only valid while the IVEK can accept Production.
        // Permanent IVEK health problems return immediately to Stopped.
        // A short ReadyProduction transient is debounced by the same timer
        // used in Manual/AutoCycle.
        IF fbIvek.IsFaulted()
            OR tonIvekCommunicationStop.Q
            OR tonIvekReferenceStop.Q
            OR tonIvekUnexpectedNotReady.Q
        THEN
            eMachineState := E_MachineState.Stopped;
        END_IF

		eMode_LED_Start := E_LEDs_Mode.FLASHING;
		eMode_LED_Reset := E_LEDs_Mode.OFF;
		eMode_LED_PASS  := E_LEDs_Mode.OFF;
		eMode_LED_Fail  := E_LEDs_Mode.OFF;
		
		
		tonInitialising(IN := FALSE);
		tonStopping(IN := FALSE);
		
		// ---------------------------------------------------------
		// PRESSURE RANGE SUPERVISION
		// ---------------------------------------------------------
		// In ReadyToStart, invalid pressure is a configuration
		// condition, not a machine fault.
		
		IF NOT stSiliconeSupplyStatus.bSiliconePressureOk
			OR NOT stSiliconeSupplyStatus.bNozzlePressureOk
		THEN
		
			IF (stInputs.rSiliconePressureBar < GVL_Config.stMachine.stSiliconeSupply.rSiliconePressureMin)
				OR (stInputs.rSiliconePressureBar > GVL_Config.stMachine.stSiliconeSupply.rSiliconePressureMax)
			THEN
				bSiliconePressureConfigRequired := TRUE;
			END_IF
		
			IF (stInputs.rNozzlePressureBar < GVL_Config.stMachine.stSiliconeSupply.rNozzlePressureMin)
				OR (stInputs.rNozzlePressureBar > GVL_Config.stMachine.stSiliconeSupply.rNozzlePressureMax)
			THEN
				bNozzlePressureConfigRequired := TRUE;
			END_IF
		
			bStopRequested := TRUE;
		
		END_IF
		
	
		IF bStopRequested THEN
	
			eMachineState := E_MachineState.Stopping;

		ELSIF stCommand.bManualRequest
			AND stInputs.stSafety.bSafetyOk
			AND NOT stIndexStatus.bBusy
			AND NOT fbIndex.IsFaulted()
			//AND NOT fbProcessStation.IsFaulted()
			//AND NOT ipEquipment.IsFaulted()
		THEN
	
			fbManualMode.Initialise();
			eMachineState := E_MachineState.Manual;
	
		ELSIF stCommand.bStart
            AND fbMainDoorLock.IsReadyForAutomatic()
            AND stSiliconeSupplyStatus.bSelectedReservoirReady
            AND bIvekAutoCycleReady
			AND NOT stInputs.bIvekHeaterControllerAlarm
			AND NOT stStatus.bIvekHeaterTemperatureOutOfRange
        THEN
	
			eCycleState := E_CycleState.Disabled;
			eMachineState := E_MachineState.AutoCycle;
	
		END_IF
// 	
	E_MachineState.AutoCycle:
		
		// ---------------------------------------------------------
		// VACUUM EXTRACTOR SUPERVISION
		// ---------------------------------------------------------
		// The extractor must remain running throughout AutoCycle.
		// Loss of feedback is an immediate machine fault because
		// the silicone process must not continue without extraction.
		// ---------------------------------------------------------
		
		IF NOT stPermissives.bExtractorReady THEN
			bExtractorAutoCycleFault := TRUE;
			bSafetyDropRequest := TRUE;
		END_IF
		
		IF stInputs.bIvekHeaterControllerAlarm OR stStatus.bIvekHeaterTemperatureOutOfRange THEN
			bSafetyDropRequest := TRUE;
		END_IF

        // Any IVEK health loss requires a controlled stop.
        IF fbIvek.IsFaulted()
            OR tonIvekCommunicationStop.Q
            OR tonIvekReferenceStop.Q
            OR tonIvekUnexpectedNotReady.Q
        THEN
            bStopRequested := TRUE;
        END_IF

		eMode_LED_Start := E_LEDs_Mode.OFF;
		eMode_LED_Reset := E_LEDs_Mode.OFF;

		// -----------------------------------------------------
		// OPERATOR RESULT LED INDICATION
		// -----------------------------------------------------
		// Same behaviour as the original implementation:
		//
		// PASS = valid result AND passed
		// FAIL = valid result AND not passed
		// -----------------------------------------------------
	
		IF stOperatorNest.stResult.bValid THEN
	
			IF stOperatorNest.stResult.bPassed THEN
	
				eMode_LED_PASS := E_LEDs_Mode.ON;
				eMode_LED_Fail := E_LEDs_Mode.OFF;
	
			ELSE
	
				eMode_LED_PASS := E_LEDs_Mode.OFF;
				eMode_LED_Fail := E_LEDs_Mode.ON;
	
			END_IF
	
		ELSE
	
			eMode_LED_PASS := E_LEDs_Mode.OFF;
			eMode_LED_Fail := E_LEDs_Mode.OFF;
	
		END_IF;

		tonInitialising(IN := FALSE);
		tonStopping(IN := FALSE);

		IF stAssemblyNest.bEnabled
			AND
			(
				stAssemblyNest.bGearboxAssemblyPartPresent
				OR stAssemblyNest.bReservoirPartPresent
			)
			AND NOT stAssemblyNest.stResult.bValid
			AND
			(
				NOT stAssemblyNest.bPartComplete
				OR NOT stAssemblyNest.stSiliconeResult.bValid
				OR NOT stAssemblyNest.stSiliconeResult.bPassed
			)
		THEN
		
			stLastResult.bValid := TRUE;
			stLastResult.bPassed := FALSE;
			stLastResult.eCode := E_ProcessResultCode.Aborted;
			stLastResult.sDetail := 'Rejected - process incomplete or Silicone not passed';
		
			bResultStoredFeedback :=
				fbNestManager.StoreResultAtPosition(
					ePosition := stConfig.eAssemblyPosition,
					stResult := stLastResult
				);
		
			IF bResultStoredFeedback THEN
		
				stAssemblyNest :=
					fbNestManager.GetNestAtPosition(
						stConfig.eAssemblyPosition
					);
		
			END_IF
		
		END_IF


	
		// PROCESS CYCLE INPUT MAPPING
		stProcessCycleInputs.bSafetyOk := stInputs.stSafety.bSafetyOk;
		stProcessCycleInputs.bTwoHandsSafe := stInputs.bTwoHandsSafe;
		
		// PROCESS REQUIREMENTS
		stProcessCycleInputs.bSiliconeProcessRequired :=
			stSiliconeNest.bEnabled
			AND stSiliconeNest.bPartComplete
			AND NOT stSiliconeNest.stResult.bValid
			AND NOT stSiliconeNest.stSiliconeResult.bValid;
		
		stProcessCycleInputs.bAssemblyProcessRequired :=
			stAssemblyNest.bEnabled
			AND stAssemblyNest.bPartComplete
			AND NOT stAssemblyNest.stResult.bValid
			AND stAssemblyNest.stSiliconeResult.bValid
			AND stAssemblyNest.stSiliconeResult.bPassed
			AND NOT stAssemblyNest.stAssemblyResult.bValid;
			
		// Indexer
		stProcessCycleInputs.bIndexPositionValid := stInputs.eIndexPosition <> E_TablePosition.Unknown;
		stProcessCycleInputs.bIndexMoveAllowed := stPermissives.bIndexMoveAllowed AND stInputs.bSiliconeSupportRetracted AND stInputs.bAssemblySupportRetracted  AND NOT stInputs.bSiliconeStationPartPresent;
		stProcessCycleInputs.bIndexReady := fbIndex.IsReady();
		stProcessCycleInputs.bIndexLocked := stInputs.bIndexLocked;
		stProcessCycleInputs.bIndexBusy := stIndexStatus.bBusy;
		stProcessCycleInputs.bIndexDone := fbIndex.IsDone();
		stProcessCycleInputs.bIndexSamePositionDetected := stIndexStatus.bSamePositionDetected;
		stProcessCycleInputs.bIndexFaulted := fbIndex.IsFaulted();
		stProcessCycleInputs.bIndexRequestAccepted := bIndexRequestAcceptedFeedback;
		stProcessCycleInputs.bIndexRecoveryRequestAccepted := bIndexRecoveryRequestAcceptedFeedback;
		
		// Silicone Support
		stProcessCycleInputs.bSiliconeSupportExtended := stInputs.bSiliconeSupportExtended;
		stProcessCycleInputs.bSiliconeSupportRetracted := stInputs.bSiliconeSupportRetracted;
		stProcessCycleInputs.bSiliconeSupportFaulted := fbSiliconeSupportCylinder.IsFaulted();
	
		// Assembly Support
		stProcessCycleInputs.bAssemblySupportExtended := stInputs.bAssemblySupportExtended;
		stProcessCycleInputs.bAssemblySupportRetracted := stInputs.bAssemblySupportRetracted;
		stProcessCycleInputs.bAssemblySupportFaulted := fbAssemblySupportCylinder.IsFaulted();
	

		stProcessCycleInputs.bOperatorExchangeComplete := fbOperatorStation.IsComplete();
	
			// =========================================================
		// SILICONE PROCESS STATUS
		// =========================================================
		
		stProcessCycleInputs.bSiliconeProcessReady 		:=fbSiliconeProcess.IsReady();
		stProcessCycleInputs.bSiliconeProcessBusy 		:=fbSiliconeProcess.IsBusy();
		stProcessCycleInputs.bSiliconeProcessComplete 	:=fbSiliconeProcess.IsDone();
		stProcessCycleInputs.bSiliconeProcessFaulted 	:=fbSiliconeProcess.IsFaulted();

		// =========================================================
		// ASSEMBLY PROCESS STATUS
		// =========================================================
		
		stProcessCycleInputs.bAssemblyProcessReady 		:=fbAssemblyStation.IsReady();
		stProcessCycleInputs.bAssemblyProcessBusy 		:=fbAssemblyStation.IsBusy();
		stProcessCycleInputs.bAssemblyProcessComplete 	:=fbAssemblyStation.IsDone();
		stProcessCycleInputs.bAssemblyProcessFaulted 	:=fbAssemblyStation.IsFaulted();
		stProcessCycleInputs.bAssemblyAtZeroPosition    :=stAssemblyStationStatus.bRotationPlace;
	
	
		// PROCESS CYCLE EXECUTION
		fbProcessCycle.Cyclic(
			bEnable := TRUE,
			bStopRequest := bStopRequested,
			bResetRequest := stCommand.bReset,
            tSequenceTimeout := stConfig.tProcessTimeout,
			stInputs := stProcessCycleInputs,
			stRequests => stProcessCycleRequests,
			stStatus => stProcessCycleStatus
		);
		
		// =========================================================
		// SILICONE PROCESS RESULT HANDLING
		// =========================================================
		
		IF fbSiliconeProcess.IsDone() THEN
		
			stLastResult := fbSiliconeProcess.GetResult();
		
			bResultStoredFeedback := fbNestManager.StoreSiliconeResultAtPosition( ePosition := stConfig.eSiliconePosition, stResult := stLastResult );
		
			IF bResultStoredFeedback THEN
				fbSiliconeProcess.RequestReset();
			END_IF
		
		END_IF
		// =========================================================
		// ASSEMBLY PROCESS RESULT HANDLING
		// =========================================================
		
		IF fbAssemblyStation.IsDone() THEN
		
			// -----------------------------------------------------
			// STORE ASSEMBLY RESULT
			// -----------------------------------------------------
		
			stLastResult := fbAssemblyStation.GetResult();
		
			bResultStoredFeedback := fbNestManager.StoreAssemblyResultAtPosition( ePosition := stConfig.eAssemblyPosition, stResult := stLastResult );
		
			IF bResultStoredFeedback THEN
		
				// -------------------------------------------------
				// READ UPDATED NEST AT ASSEMBLY POSITION
				// -------------------------------------------------
		
				stAssemblyNest := fbNestManager.GetNestAtPosition( stConfig.eAssemblyPosition );
		
				// -------------------------------------------------
				// CALCULATE FINAL RESULT
				// -------------------------------------------------
		
				stLastResult.bValid := stAssemblyNest.stSiliconeResult.bValid AND stAssemblyNest.stAssemblyResult.bValid;
		
				stLastResult.bPassed := stLastResult.bValid AND stAssemblyNest.stSiliconeResult.bPassed AND stAssemblyNest.stAssemblyResult.bPassed;
		
				// -------------------------------------------------
				// STORE FINAL RESULT IN NEST
				// -------------------------------------------------
		
				bResultStoredFeedback := fbNestManager.StoreResultAtPosition( ePosition := stConfig.eAssemblyPosition, stResult := stLastResult );
		
				// -------------------------------------------------
				// RESET ASSEMBLY PROCESS
				// -------------------------------------------------
		
				IF bResultStoredFeedback THEN
					fbAssemblyStation.RequestReset();
				END_IF
		
			END_IF
		
		END_IF
		
		// =========================================================
		// STATION PROCESS REQUEST EXECUTION
		// =========================================================
		
		// Silicone Process
		IF stProcessCycleRequests.bStartSiliconeProcess THEN
			fbSiliconeProcess.RequestStart();
		END_IF
		
		IF stProcessCycleRequests.bStopSiliconeProcess THEN
			fbSiliconeProcess.RequestStop();
		END_IF
		
		
		// Assembly Process
		IF stProcessCycleRequests.bStartAssemblyProcess THEN
			fbAssemblyStation.RequestStart();
		END_IF
		
		IF stProcessCycleRequests.bStopAssemblyProcess THEN
			fbAssemblyStation.RequestStop();
		END_IF
		
		
			//Timeout process
		tonAutoCycleIdleTimeout(
			IN := stProcessCycleStatus.eState = E_CycleState.WaitingForProcessCycleTrigger,
			PT := T#2M
		);
		
		// FEEDBACK DEFAULTS
		bIndexRequestAcceptedFeedback := FALSE;
		bIndexRecoveryRequestAcceptedFeedback := FALSE;
		// bResultStoredFeedback := FALSE;
	
		// INDEX REQUEST EXECUTION
		IF stProcessCycleRequests.bRequestIndex THEN
			bIndexRequestAcceptedFeedback := fbIndex.RequestMove();
		END_IF
	
		IF stProcessCycleRequests.bRequestIndexRecovery THEN
			bIndexRecoveryRequestAcceptedFeedback := fbIndex.RequestPositionRecovery();
		END_IF
	
		// FUTURE PROCESS REQUEST EXECUTION
		// IF stProcessCycleRequests.bStartProcessStation THEN
		//     fbIvek.RequestStart();
		// END_IF
	
		// IF stProcessCycleRequests.bStopProcessStation THEN
		//     fbIvek.RequestStop();
		// END_IF
	
		// IF stProcessCycleRequests.bCaptureProcessResult THEN
		//     stLastResult := fbProcessStation.GetResult();
		// END_IF
	
		// IF stProcessCycleRequests.bStoreProcessResult THEN
		//     stLastResult := fbProcessStation.GetResult();
		//     bResultStoredFeedback := fbNestManager.StoreResultAtPosition(
		//         ePosition := stConfig.eProcessPosition,
		//         stResult := stLastResult
		//     );
		//
		//     IF bResultStoredFeedback THEN
		//         fbIndex.ReleaseProcessPosition();
		//     END_IF
		// END_IF
	
		// IF stProcessCycleRequests.bConfirmOperatorExchange THEN
		//     fbNestManager.MarkDispositionComplete(stConfig.eOperatorPosition);
		//     fbIndex.ConfirmOperatorExchange();
		// END_IF
	
		// IF stProcessCycleRequests.bUpdateNestPositions THEN
		//     fbNestManager.ClearOperatorNest(stConfig.eOperatorPosition);
		// END_IF
	
		// PROCESS CYCLE FAULT
		IF stProcessCycleStatus.bFaulted THEN
			bSafetyDropRequest := TRUE;
		END_IF
	
		// LEAVE AUTO CYCLE
		IF bStopRequested
			AND stProcessCycleStatus.eState = E_CycleState.Disabled
		THEN
			eMachineState := E_MachineState.Stopping;
		END_IF
		
		IF tonAutoCycleIdleTimeout.Q THEN
			 bStopRequested := TRUE;
		END_IF
// 	
	E_MachineState.Manual:


        // Manual follows the same IVEK health interlock.
        IF fbIvek.IsFaulted()
            OR tonIvekCommunicationStop.Q
            OR tonIvekReferenceStop.Q
            OR tonIvekUnexpectedNotReady.Q
        THEN
            bStopRequested := TRUE;
        END_IF

		eMode_LED_Start := E_LEDs_Mode.OFF;
		eMode_LED_Reset := E_LEDs_Mode.OFF;
		eMode_LED_PASS  := E_LEDs_Mode.OFF;
		eMode_LED_Fail  := E_LEDs_Mode.OFF;
		
		tonInitialising(IN := FALSE);
		tonStopping(IN := FALSE);
		
		// ---------------------------------------------------------
		// INDEX MANUAL MOVEMENT
		// ---------------------------------------------------------
		IF stManualModeRequests.bIndexMoveRequest THEN
	
			bManualIndexRequestAccepted := fbIndex.RequestManualMove();
	
		END_IF
	
	
		// ---------------------------------------------------------
		// INDEX RESET / HOME
		// ---------------------------------------------------------
		// At this stage the home command resets the pneumatic index sequence.
		// A dedicated homing method can be introduced later if required.
		IF stManualModeRequests.bIndexHomeRequest THEN
	
			fbIndex.Reset();
	
		END_IF
	
	
		// ---------------------------------------------------------
		// MANUAL SILICONE PROCESS
		// ---------------------------------------------------------
		IF stManualModeRequests.bSiliconeProcessStart THEN
			bManualSiliconeCycleActive := TRUE;
		END_IF
		
		// Start the Silicone Process only after the support
		// has reached the extended position.
		IF bManualSiliconeCycleActive
			AND stInputs.bSiliconeSupportExtended
			AND fbSiliconeProcess.IsReady()
		THEN
			fbSiliconeProcess.RequestStart();
END_IF

		IF stManualModeRequests.bSiliconeProcessStop THEN
			fbSiliconeProcess.RequestStop();
		END_IF

		IF bManualSiliconeCycleActive
			AND fbSiliconeProcess.IsDone()
		THEN
		
			stLastResult := fbSiliconeProcess.GetResult();
		
			bResultStoredFeedback :=
				fbNestManager.StoreSiliconeResultAtPosition(
					ePosition := stConfig.eSiliconePosition,
					stResult := stLastResult
				);
		
		END_IF
		
		
		IF bManualSiliconeCycleActive
			AND fbSiliconeProcess.IsDone()
			AND stInputs.bSiliconeSupportRetracted
		THEN
		
			fbSiliconeProcess.RequestReset();
			bManualSiliconeCycleActive := FALSE;
		
		END_IF

		// ---------------------------------------------------------
		// PROCESS EQUIPMENT MANUAL COMMANDS
		// ---------------------------------------------------------
		IF stManualModeRequests.bEquipmentStart
		AND NOT bManualSiliconeCycleActive THEN

			fbIvek.RequestStart();

		END_IF
	
		IF stManualModeRequests.bEquipmentStop
		AND NOT bManualSiliconeCycleActive THEN

			fbIvek.RequestStop();

		END_IF
	
		IF stManualModeRequests.bEquipmentReset
		AND NOT bManualSiliconeCycleActive THEN

			fbIvek.RequestReset();

		END_IF
	
		// ---------------------------------------------------------
		// LEAVE MANUAL MODE
		// ---------------------------------------------------------
		//
		// The Manual Mode coordinator first returns all manually
		// controlled components to their standard state.
		//
		// Machine state may leave Manual only after the coordinator
		// confirms that the exit sequence is complete.
		// ---------------------------------------------------------
		
		IF bStopRequested
			AND stManualModeStatus.bSafeToExit
		THEN
			eMachineState := E_MachineState.Stopping;
		END_IF
		
END_CASE



// =========================================================
// PROCESS CYCLE DISABLE HANDLING
// =========================================================
IF eMachineState <> E_MachineState.AutoCycle THEN
	fbProcessCycle.Cyclic(
        bEnable := FALSE,
        bResetRequest := stCommand.bReset,
        bStopRequest := TRUE,
        tSequenceTimeout := stConfig.tProcessTimeout,
        stInputs := stProcessCycleInputs,
        stRequests =>stProcessCycleRequests,
        stStatus =>stProcessCycleStatus);
END_IF

    

// =========================================================
// CYCLIC COMPONENT EXECUTION
// =========================================================
// =========================================================
// SUPPORT COMMAND SELECTION
// =========================================================

bSiliconeSupportRaiseRequest := FALSE;
bSiliconeSupportLowerRequest := FALSE;
bAssemblySupportRaiseRequest := FALSE;
bAssemblySupportLowerRequest := FALSE;


// ---------------------------------------------------------
// INITIALISING
// ---------------------------------------------------------
// Return both process supports to their standard
// safe retracted position before ReadyToStart.
// ---------------------------------------------------------

IF eMachineState = E_MachineState.Initialising THEN

    // Supports may only be recovered after the pneumatic
    // supply has been confirmed by TwinSAFE.
    IF stPermissives.bAirSupplyReady THEN

        bSiliconeSupportLowerRequest := TRUE;
        bAssemblySupportLowerRequest := TRUE;

    END_IF


// ---------------------------------------------------------
// MANUAL MODE
// ---------------------------------------------------------

ELSIF eMachineState = E_MachineState.Manual THEN
	
	IF bManualSiliconeCycleActive THEN
	
		IF fbSiliconeProcess.IsDone() THEN
	
			bSiliconeSupportRaiseRequest := FALSE;
			bSiliconeSupportLowerRequest := TRUE;
	
		ELSE
	
			bSiliconeSupportRaiseRequest := TRUE;
			bSiliconeSupportLowerRequest := FALSE;
	
		END_IF
	
	ELSE
	
		bSiliconeSupportRaiseRequest :=
			stManualModeRequests.bSiliconeSupportExtend;
	
		bSiliconeSupportLowerRequest :=
			stManualModeRequests.bSiliconeSupportRetract;
	
	END_IF

	IF bManualAssemblyCycleActive THEN

		// During the active flipping sequence:
		// 180 -> 0 with support down.
		// At 0°, raise support and keep it raised.
		// Once the Assembly Station completes, retract the support.
		IF fbAssemblyStation.IsDone() THEN
	
			bAssemblySupportRaiseRequest := FALSE;
			bAssemblySupportLowerRequest := TRUE;
	
		ELSE
	
			bAssemblySupportRaiseRequest :=
				stAssemblyStationStatus.bRotationPlace
				OR stInputs.bAssemblySupportExtended;
	
			bAssemblySupportLowerRequest := FALSE;
	
		END_IF
	
	ELSE
	
		// Normal Manual Mode support control.
		bAssemblySupportRaiseRequest :=
			stManualModeRequests.bAssemblySupportExtend;
	
		bAssemblySupportLowerRequest :=
			stManualModeRequests.bAssemblySupportRetract;
	
	END_IF

    // Manual assembly/flipping request execution.
	IF stManualModeRequests.bAssemblyStationStart THEN
		IF fbAssemblyStation.RequestStart() THEN
			bManualAssemblyCycleActive := TRUE;
		END_IF
	END_IF

    IF stManualModeRequests.bAssemblyStationStop THEN
        fbAssemblyStation.RequestStop();
    END_IF




//     // ---------------------------------------------------------
//     // MANUAL ASSEMBLY RESULT HANDLING
//     // ---------------------------------------------------------
//     // A manual "Assemble Parts" action is a real process operation. Store its
//     // assembly result at the nest currently mapped to the Assembly Station so
//     // the same part will not be flipped again after returning to AutoCycle.
//     IF bManualAssemblyCycleActive AND fbAssemblyStation.IsDone() THEN
// 
//         stLastResult := fbAssemblyStation.GetResult();
// 
//         bResultStoredFeedback :=
//             fbNestManager.StoreAssemblyResultAtPosition(
//                 ePosition := stConfig.eAssemblyPosition,
//                 stResult := stLastResult
//             );
// 
//         IF bResultStoredFeedback THEN
// 
//             stAssemblyNest :=
//                 fbNestManager.GetNestAtPosition(stConfig.eAssemblyPosition);
// 
//             stLastResult.bValid :=
//                 stAssemblyNest.stSiliconeResult.bValid
//                 AND stAssemblyNest.stAssemblyResult.bValid;
// 
//             stLastResult.bPassed :=
//                 stLastResult.bValid
//                 AND stAssemblyNest.stSiliconeResult.bPassed
//                 AND stAssemblyNest.stAssemblyResult.bPassed;
// 
//             bResultStoredFeedback :=
//                 fbNestManager.StoreResultAtPosition(
//                     ePosition := stConfig.eAssemblyPosition,
//                     stResult := stLastResult
//                 );
// 
//             IF bResultStoredFeedback THEN
//                 fbAssemblyStation.RequestReset();
//                 bManualAssemblyCycleActive := FALSE;
//             END_IF
// 
//         END_IF
// 
//     END_IF


	IF bManualAssemblyCycleActive
		AND fbAssemblyStation.IsDone()
		AND stInputs.bAssemblySupportRetracted
	THEN
		fbAssemblyStation.RequestReset();
		bManualAssemblyCycleActive := FALSE;
	END_IF


// ---------------------------------------------------------
// AUTOMATIC CYCLE
// ---------------------------------------------------------

ELSIF eMachineState = E_MachineState.AutoCycle THEN

    bSiliconeSupportRaiseRequest := stProcessCycleRequests.bSiliconeSupportExtend;
    bSiliconeSupportLowerRequest := stProcessCycleRequests.bSiliconeSupportRetract;

    bAssemblySupportRaiseRequest := stProcessCycleRequests.bAssemblySupportExtend;
    bAssemblySupportLowerRequest := stProcessCycleRequests.bAssemblySupportRetract;

END_IF



// =========================================================
// ASSEMBLY / FLIPPING STATION CONTROL
// =========================================================
// Physical mapping from EPLAN Rev 1.0:
//   Term 8 Ch5..10  = slide, gripper and rotation feedback
//   Term 10 Ch9..14 = slide, gripper and rotation valve commands
//
// During Initialising the object automatically returns to:
//   slide retracted + gripper open + rotation 0 degrees.
// During AutoCycle it executes the complete barrel pick/flip/place sequence.
// =========================================================

fbAssemblyStation.Cyclic(
    bEnable :=
        (eMachineState = E_MachineState.AutoCycle)
        OR
        (
            (eMachineState = E_MachineState.Manual)
            AND stCommand.bAssemblyStationManualEnable
        ),
    bInitialising := (eMachineState = E_MachineState.Initialising),
    bSafetyPermitted := stInputs.stSafety.bProcessSafetyPermitted,
    bAirSupplySafe := stPermissives.bAirSupplyReady,
    bIndexReady := stInputs.bIndexReady,
    bIndexLocked := stInputs.bIndexLocked,
    bIndexBusy := stIndexStatus.bBusy,
    bAssemblySupportExtended := stInputs.bAssemblySupportExtended,
    bSlideExtended := stInputs.bTransferVerticalMiniSlideExtended,
    bSlideRetracted := stInputs.bTransferVerticalMiniSlideRetracted,
    bGripperOpen := stInputs.bRotaryGripperOpened,
    bGripperClosed := stInputs.bRotaryGripperClosed,
    bRotationPick := stInputs.bRotaryGripperRotationPick0,
    bRotationPlace := stInputs.bRotaryGripperRotationPlace180,
    tActionDelay := stConfig.tAssemblyActionDelay,
    tMovementTimeout := stConfig.tAssemblyMovementTimeout,
	tReleaseDelay := stConfig.tAssemblyReleaseDelay,
    bSlideExtendOutput => stOutputsInternal.bTransferVerticalMiniSlideExtend,
    bSlideRetractOutput => stOutputsInternal.bTransferVerticalMiniSlideRetract,
    bGripperOpenOutput => stOutputsInternal.bRotaryGripperOpen,
    bGripperCloseOutput => stOutputsInternal.bRotaryGripperClose,
    bRotationPickOutput => stOutputsInternal.bRotaryGripperRotationPick0,
    bRotationPlaceOutput => stOutputsInternal.bRotaryGripperRotationPlace180
);

stAssemblyStationStatus := fbAssemblyStation.GetStatus();

// =========================================================
// SILICONE SUPPORT CONTROL
// =========================================================

fbSiliconeSupportCylinder.Cyclic(
	bEnable := (eMachineState = E_MachineState.Initialising)
				OR (eMachineState = E_MachineState.Manual)
				OR (eMachineState = E_MachineState.AutoCycle),
    bRaiseRequest := bSiliconeSupportRaiseRequest,
    bLowerRequest := bSiliconeSupportLowerRequest,
    bStopRequest := (eMachineState = E_MachineState.Stopping)
        OR (eMachineState = E_MachineState.Fault),
    bExtended := stInputs.bSiliconeSupportExtended,
    bRetracted := stInputs.bSiliconeSupportRetracted,
    tMovementTimeout := stConfig.tCylinderTimeout,
    bExtendOutput => stOutputsInternal.bSiliconeSupportExtend,
    bRetractOutput => stOutputsInternal.bSiliconeSupportRetract
);

// =========================================================
// ASSEMBLY SUPPORT CONTROL
// =========================================================

fbAssemblySupportCylinder.Cyclic(
	bEnable := (eMachineState = E_MachineState.Initialising)
				OR (eMachineState = E_MachineState.Manual)
				OR (eMachineState = E_MachineState.AutoCycle),
    bRaiseRequest := bAssemblySupportRaiseRequest,
    bLowerRequest := bAssemblySupportLowerRequest,
    bStopRequest := (eMachineState = E_MachineState.Stopping)
        OR (eMachineState = E_MachineState.Fault),
    bExtended := stInputs.bAssemblySupportExtended,
    bRetracted := stInputs.bAssemblySupportRetracted,
    tMovementTimeout := stConfig.tCylinderTimeout,
    bExtendOutput => stOutputsInternal.bAssemblySupportExtend,
    bRetractOutput => stOutputsInternal.bAssemblySupportRetract
);


// ---------------------------------------------------------
// INITIALISING - FORCE SUPPORTS RETRACT PRESSURE
// ---------------------------------------------------------
// Keep both retract valves energised during Initialising,
// regardless of the retracted feedback. This pre-pressurises
// the retract side before the first automatic extension.
// ---------------------------------------------------------

IF (eMachineState = E_MachineState.Initialising)
    AND stPermissives.bAirSupplyReady
THEN

    stOutputsInternal.bSiliconeSupportExtend := FALSE;
    stOutputsInternal.bSiliconeSupportRetract := TRUE;

    stOutputsInternal.bAssemblySupportExtend := FALSE;
    stOutputsInternal.bAssemblySupportRetract := TRUE;

END_IF


// Cyclic component execution
// LEGACY PROCESS STATION:
// Do not execute FB_ProcessStation in Manual mode. Its legacy Manual branch
// calls ipEquipment.RequestStop() continuously, which conflicts with the
// new FB_SiliconeProcess -> FB_IvekDigiSpense4000 manual runtime path.
IF eMachineState <> E_MachineState.Manual THEN

fbProcessStation.Cyclic(
    bEnable :=
    (eMachineState = E_MachineState.Initialising)
    OR
    (eMachineState = E_MachineState.AutoCycle),
    bAutomaticStartRequest 			:= bProcessStartPulse,
    bManualEnable 					:= eMachineState = E_MachineState.Manual,
	bAirSupplySafe 					:= GVL_Safety.bAirSupplySafe,
    bManualExtendRequest 			:= FALSE,
    bManualRetractRequest 			:= FALSE,
    bStopRequest 					:= (eMachineState = E_MachineState.Stopping) OR (eMachineState = E_MachineState.Fault),
    bResetRequest 					:= stCommand.bReset,
    bPartPresent					:= stInputs.bReservoirPartPresent,
    bProcessPermissive 				:= stPermissives.bProcessStartAllowed,
    bIndexReady 					:= stInputs.bIndexReady,
    bIndexLocked 					:= stInputs.bIndexLocked,
    bIndexBusy 						:= stIndexStatus.bBusy,
    bProcessSafetyPermitted 		:= stInputs.stSafety.bProcessSafetyPermitted,
    bMainDoorSafe 					:= stInputs.stSafety.bMainDoorSafe,
    bCylinderExtended 				:= stInputs.bSiliconeSupportExtended,
    bCylinderRetracted 				:= stInputs.bSiliconeSupportRetracted,
    tCylinderTimeout 				:= stConfig.tCylinderTimeout,
    tProcessTimeout 				:= stConfig.tProcessTimeout,
    bCylinderExtendOutput 			=> bProcExtend,
    bCylinderRetractOutput 			=> bProcRetract
);

END_IF


// =========================================================
// MAIN DOOR LOCK CONTROL
// =========================================================

fbMainDoorLock.Cyclic(
    bEnableAutomatic := bAirAndDoorEnable,

    bManualEnable := FALSE,
    bManualLockRequest := FALSE,
    bManualUnlockRequest := FALSE,

    bStopRequest :=
        (eMachineState = E_MachineState.Fault)
        OR (eMachineState = E_MachineState.Stopping)
        OR (eMachineState = E_MachineState.Stopped),

    bResetRequest := stCommand.bReset,

    bDoorClosed := stInputs.bMainDoorClosed,
	bDoorLocked := stInputs.bMainDoorLocked,
	bDoorUnsafe := stInputs.bMainDoorUnsafe,

    bIndexBusy := stIndexStatus.bBusy,
    bProcessSafePosition := fbProcessStation.IsSafePosition() AND fbAssemblyStation.IsHome(),

    tLockTimeout := GVL_config.stMachine.tDoorLockTimeout,
    tUnlockTimeout := GVL_config.stMachine.tDoorUnlockTimeout
);

stMainDoorLockStatus := fbMainDoorLock.GetStatus();

// The standard PLC only requests that the door be locked.
// TwinSAFE validates the safe conditions and controls the physical locker.
stOutputsInternal.bMainDoorLockRequest := bAirAndDoorEnable;

// =========================================================
// INDEX TABLE CONTROL
// =========================================================
fbIndex.Cyclic(
    bEnable := (eMachineState = E_MachineState.Initialising)
        OR (eMachineState = E_MachineState.ReadyToStart)
        OR (eMachineState = E_MachineState.AutoCycle)
        OR (eMachineState = E_MachineState.Manual)
        OR (eMachineState = E_MachineState.Stopping),
    bReset := stCommand.bReset,
    bAutomaticMode := eMachineState = E_MachineState.AutoCycle,
    bManualMode := eMachineState = E_MachineState.Manual,
    bMovePermissive :=
    (
        (eMachineState = E_MachineState.AutoCycle)
        AND stInputs.bSiliconeSupportRetracted
        AND stInputs.bAssemblySupportRetracted
        AND fbAssemblyStation.IndexPermissive()
        AND
        (
            stPermissives.bIndexMoveAllowed
            OR
            (
                (stInputs.eIndexPosition = E_TablePosition.Unknown)
                AND stInputs.stSafety.bMotionSafetyPermitted
            )
        )
    )
    OR
    (
        stManualModeStatus.bIndexPermissive
        AND (eMachineState = E_MachineState.Manual)
    ),
    bSafetyMotionPermitted := stInputs.stSafety.bMotionSafetyPermitted,
    bTwoHandsSafe := stInputs.bTwoHandsSafe,
    bStationsHome := stInputs.bSiliconeSupportRetracted
        AND stInputs.bAssemblySupportRetracted
        AND fbAssemblyStation.IsHome(),
    bProcessToolingRetracted := stInputs.bSiliconeSupportRetracted
        AND stInputs.bAssemblySupportRetracted
        AND fbAssemblyStation.IsHome(),
    bTableReady := stInputs.bIndexReady,
    bTableLocked := stInputs.bIndexLocked,
    bCompletedSensor := stInputs.bIndexCompletedSensor,
    bSupportExtended := stInputs.bIndexSupportExtended,
    bSupportRetracted := stInputs.bIndexSupportRetracted,
    eCurrentPosition := stInputs.eIndexPosition,
    tRotateDelay := stConfig.tIndexRotateDelay,
    tStopDelay := stConfig.tIndexStopDelay,
    tSupportTimeout := stConfig.tIndexSupportTimeout,
    tMovementTimeout := stConfig.tIndexTimeout,
    tTwoHandHold := stConfig.tTwoHandHold,
    tTwoHandRecoveryTimeout := stConfig.tTwoHandRecoveryTimeout,
    bRotatePortA => stOutputsInternal.bIndexRotatePortA,
    bStopPortB => stOutputsInternal.bIndexStopPortB,
    bSupportExtendRequest => stOutputsInternal.bIndexSupportExtend,
    bSupportRetractRequest => stOutputsInternal.bIndexSupportRetract);
	

// =========================================================
// COMPONENT FAULT AGGREGATION
// =========================================================
	CheckComponentFaults();

// =========================================================
// PLC FAULT TO TWINSAFE RUN-DROP PULSE
// =========================================================

// Convert the one-scan internal request into a timed TwinSAFE run drop.
// This block must execute after the machine-state logic because fault
// transitions inside the CASE generate bSafetyDropRequest.
tpSafetyRunDrop(
    IN := bSafetyDropRequest,
    PT := T#500MS
);


// =========================================================
// EVENT-DRIVEN MACHINE TRANSITIONS
// =========================================================

// IF stInputs.bEventFault THEN
//     eMachineState := E_MachineState.Fault;
// ELSIF stInputs.bEventCycleStopRequest
//       AND (eMachineState = E_MachineState.AutoCycle OR eMachineState = E_MachineState.Manual)
// THEN
//     eMachineState := E_MachineState.Stopping;
// END_IF

// =========================================================
// MACHINE OUTPUT MAPPING
// =========================================================

// Outputs and public status
stOutputsInternal.bAirSupplyEnable := bAirSupplyEnable;
// An internal PLC machine fault temporarily removes the TwinSAFE run request.
// The request returns automatically after the configured TP duration.
stOutputsInternal.bSafetyRunRequest := NOT tpSafetyRunDrop.Q;
//stOutputsInternal.bSafetyRunRequest := TRUE;
stOutputsInternal.bSafetyResetRequest := stCommand.bReset AND NOT stInputs.stSafety.bSafetyOk;

stOutputsInternal.bSafetyErrorAcknowledgementRequest :=stOutputsInternal.bSafetyResetRequest;

// stOutputsInternal.bLedStart 		:= eMachineState = E_MachineState.ReadyToStart;
// stOutputsInternal.bLedReset 		:= eMachineState = E_MachineState.Fault OR eMachineState = E_MachineState.Stopped;
// // Result LEDs represent only the part currently
// // located at the operator position.
// stOutputsInternal.bLedPass 			:= stOperatorNest.stResult.bValid AND stOperatorNest.stResult.bPassed;
// stOutputsInternal.bLedFail 			:= (stOperatorNest.stResult.bValid AND NOT stOperatorNest.stResult.bPassed) OR eMachineState = E_MachineState.Fault;
stOutputsInternal.bInternalLight 	:= NOT stInputs.bMainDoorClosed;
stOutputsInternal.bExternalLight 	:= stCommand.bExternalLight;
stOutputsInternal.bExtractorEnable  := bExtractorEnable;


// =========================================================
// LED OUTPUT MAPPING
// =========================================================
	
	// START LED
	CASE eMode_LED_Start OF
		
		E_LEDs_Mode.OFF:stOutputsInternal.bLedStart := FALSE;
		E_LEDs_Mode.ON:stOutputsInternal.bLedStart := TRUE;
		E_LEDs_Mode.FLASHING:stOutputsInternal.bLedStart := bLedBlink;
	
	END_CASE
	// RESET LED
	CASE eMode_LED_Reset OF
	
		E_LEDs_Mode.OFF:stOutputsInternal.bLedReset := FALSE;
		E_LEDs_Mode.ON:stOutputsInternal.bLedReset := TRUE;
		E_LEDs_Mode.FLASHING:stOutputsInternal.bLedReset := bLedBlink;
	
	END_CASE
	// PASS LED
	CASE eMode_LED_PASS OF
	
		E_LEDs_Mode.OFF:stOutputsInternal.bLedPass := FALSE;
		E_LEDs_Mode.ON:stOutputsInternal.bLedPass := TRUE;
		E_LEDs_Mode.FLASHING:stOutputsInternal.bLedPass := bLedBlink;
	
	END_CASE	
	// FAIL LED
	CASE eMode_LED_Fail OF
		E_LEDs_Mode.OFF:stOutputsInternal.bLedFail := FALSE;
		E_LEDs_Mode.ON:stOutputsInternal.bLedFail := TRUE;
		E_LEDs_Mode.FLASHING:stOutputsInternal.bLedFail := bLedBlink;
	
	END_CASE


// =========================================================
// EQUIPMENT OUTPUT DATA
// =========================================================

stIvekOutput := fbIvek.stCyclicOut;
// =========================================================
// PUBLIC MACHINE STATUS
// =========================================================

stStatus.eMachineState 			:= eMachineState;
stStatus.eCycleState 			:= stProcessCycleStatus.eState;
stStatus.stProcessCycle 		:= stProcessCycleStatus;
stStatus.stProcessStation 		:= stProcessStationStatus;
stStatus.stAssemblyStation      := stAssemblyStationStatus;
stStatus.bDisabledNestPartPresent := bDisabledNestPartPresent;

// Manual HMI projection for the physical Silicone Station.
stStatus.uiSiliconeStationNestId := stSiliconeNest.nId;
stStatus.bSiliconeStationPartPresent :=stInputs.bSiliconeStationPartPresent;
stStatus.bSiliconeStationReady :=
    stManualModeStatus.bSiliconeStationStartPermissive;
stStatus.bSiliconeStationManualEnabled :=
    (eMachineState = E_MachineState.Manual)
    AND stCommand.bSiliconeStationManualEnable;
stStatus.bSiliconeStationManualStartPermissive :=
    stManualModeStatus.bSiliconeStationStartPermissive;



// Positive IVEK status booleans for TRUE=green / FALSE=red HMI convention.
stStatus.bIvekReady := fbIvek.IsReady();
stStatus.bIvekProductionReady := fbIvek.bReadyProduction;
stStatus.bIvekBusy := fbIvek.IsBusy();
stStatus.bIvekHealthy := bIvekCommsOk AND NOT fbIvek.IsFaulted();
stStatus.bIvekFaulted := fbIvek.IsFaulted();
stStatus.bIvekMotionEnabled := bIvekCommsOk AND NOT fbIvek.bMotionDisabled;
stStatus.bIvekReferenceRequired := fbIvek.IsReferenceRequired();
stStatus.bIvekReferenceReady := fbIvek.bReadyReference;
stStatus.bIvekReferenceActive := fbIvek.IsReferenceActive();
stStatus.bIvekFluidicReady := fbIvek.IsFluidicReady();
stStatus.bIvekFluidicActive := fbIvek.IsFluidicActive();

stStatus.bIvekPrimePermissive :=
    stManualModeStatus.bIvekPrimePermissive;
	
stStatus.bIvekReferencePermissive :=
    bIvekMaintenancePermissive
    AND fbIvek.IsReferenceRequired()
    AND fbIvek.bReadyReference;

// Manual HMI projection for the physical Assembly Station.
stStatus.uiAssemblyStationNestId := stAssemblyNest.nId;
stStatus.bAssemblyStationPartPresent := stAssemblyNest.bPartComplete;
stStatus.bAssemblyStationPartSiliconized :=
    stAssemblyNest.stSiliconeResult.bValid
    AND stAssemblyNest.stSiliconeResult.bPassed;
stStatus.bAssemblyStationManualEnabled :=
    (eMachineState = E_MachineState.Manual)
    AND stCommand.bAssemblyStationManualEnable;
stStatus.bAssemblyStationManualStartPermissive :=
    stManualModeStatus.bAssemblyStationStartPermissive;
stStatus.stMainDoorLock 		:= stMainDoorLockStatus;
stStatus.eInitialisingWaitReason := eInitialisingWaitReason;
stStatus.eStoppingWaitReason 	:= eStoppingWaitReason;
stIndexStatus 					:= fbIndex.GetStatus();
stStatus.eIndexState 			:= stIndexStatus.eState;
stStatus.stIndexStatus 			:= stIndexStatus;
stStatus.eEquipmentState 		:= ipEquipment.GetState();
stStatus.eOperatorExchangeState := fbOperatorStation.GetState();
stStatus.eOperatorInstruction 	:= fbOperatorStation.GetInstruction();
stStatus.stOperatorStation 		:= stOperatorStatus;
stStatus.eManualModeState 		:= stManualModeStatus.eState;
stStatus.stManualMode 			:= stManualModeStatus;
stStatus.bReady 				:= eMachineState = E_MachineState.ReadyToStart;
stStatus.bBusy 					:= eMachineState = E_MachineState.AutoCycle;
stStatus.bFaulted 				:= eMachineState = E_MachineState.Fault;
stStatus.bInitialisationTimeoutFault := bInitialisationTimeoutFault;
stStatus.bExtractorAutoCycleFault := bExtractorAutoCycleFault;
stStatus.bHmiLogoutFault 		:= bHmiLogoutFault;
stStatus.bStoppingTimeoutFault 	:= bStoppingTimeoutFault;
stStatus.bSafetyStopRequested 	:= tpSafetyRunDrop.Q;
stStatus.bSafetyRunRequested 	:= stOutputsInternal.bSafetyRunRequest;
stStatus.bEventFault 			:= stInputs.bEventFault;
stStatus.bStopRequestTimeout 	:= bStopRequestTimeout;

stStatus.bIndexPermissive 		:= stPermissives.bIndexMoveAllowed;
stStatus.bProcessPermissive 	:= stPermissives.bProcessStartAllowed;
stStatus.stPermissives 			:= stPermissives;
stStatus.stLastResult 			:= stLastResult;
stStatus.bEnableSetting 		:= eMachineState = E_MachineState.Stopped;
GVL_Persistent.stStatistics.aNest := fbNestManager.GetAllNestStatistics();
stStatus.bSiliconeSupportFaulted := fbSiliconeSupportCylinder.IsFaulted();
stStatus.bAssemblySupportFaulted := fbAssemblySupportCylinder.IsFaulted();
stStatus.bAssemblyStationFaulted := fbAssemblyStation.IsFaulted();
stStatus.bPartVacuumBuildTimeoutFault :=fbSiliconeProcess.bVacuumBuildTimeoutFault;
stStatus.bPartVacuumLostFault :=fbSiliconeProcess.bVacuumLostFault;
stStatus.bPartVacuumReleaseTimeoutFault :=fbSiliconeProcess.bVacuumReleaseTimeoutFault;
stStatus.bSiliconePressureFault := bSiliconePressureFault;
stStatus.bNozzlePressureFault := bNozzlePressureFault;
stStatus.bSiliconePressureConfigRequired := bSiliconePressureConfigRequired;
stStatus.bNozzlePressureConfigRequired := bNozzlePressureConfigRequired;


stCycleDataCSVOut := stCycleDataCSV;
bCycleDataCSVWriteOut := bCycleDataCSVWrite;

